// TIA Portal project "SimLogic" (V15)

(* hardware
DEVICE "S71500/ET200MP station_1"  S7-1500 station
   slot 0: "Rail_0"  Rack  6ES7 590-1***0-0AA0
   slot 1: "PLC_1"  CPU 1511-1 PN  6ES7 511-1AK00-0AB0  V1.8
      slot 3: "CPU display_1"  6ES7591-1AA00-0AA0
DEVICE "PC-System_1"  SIMATIC PC station
   slot 0: "SIMATIC PC station"  Rail  SIMATIC PC-Station  V1.0
      slot 125: "Stationmanager"  Station_Manager  V6.0.4
   slot 1: "HMI_RT_1"  WinCC RT Advanced  6AV2 104-0xxxx-xxxx  15.0.0.0
      slot 33792: "Host interface"  Host interface
   slot 2: "IE general_1"  IE General  IE_CP  V8.2.0
*)

// ===== PLC "PLC_1"  CPU 1511-1 PN =====

VAR_GLOBAL   // PLC tag table "Default tag table"
   "Brake_Out" AT %M0.0 : Bool;
   "Baffle_Out" AT %MW18 : Int;
   "RPM_In" AT %MW2 : Int;
   "OilTemp_In" AT %MW4 : Int;
   "Baffle_En" AT %M0.1 : Bool;
   "Current_In" AT %MW6 : Int;
   "OilPumpVFDsp_Out" AT %MW8 : Int;
   "OilPumpVFDen_Out" AT %M0.2 : Bool;
   "OilFlow_In" AT %MW10 : Int;
   "PB_LAD" AT %M0.3 : Bool;
   "ONS" AT %M0.4 : Bool;
   "PROGLANG" AT %MW12 : Int;
   "ONS3" AT %M0.5 : Bool;
   "ONS2" AT %M0.6 : Bool;
   "ONS1" AT %M0.7 : Bool;
   "PB_FBD" AT %M1.0 : Bool;
   "PB_SCL" AT %M1.1 : Bool;
   "PB_STL" AT %M1.2 : Bool;
   "AlarmHorn_out" AT %M1.3 : Bool;
   "stationInterlock_out" AT %M1.4 : Bool;
   "input_max" AT %MD14 : DInt;
   "OilpumpVFD_pct" AT %MW20 : Int;
   "baffle_pct" AT %MW22 : Int;
   "OiltempSV" AT %MW24 : Int;
   "OilflowSV" AT %MW26 : Int;
   "RPMout_SV" AT %MW28 : Int;
   "curentout_SV" AT %MW30 : Int;
   "oilpumpVFDoff_pb" AT %M1.5 : Bool;
   "oilpumpVFDon_pb" AT %M1.6 : Bool;
   "oilpumpVFDauto_pb" AT %M1.7 : Bool;
   "brakeoff_pb" AT %M34.0 : Bool;
   "brakeon_pb" AT %M34.1 : Bool;
   "brakeauto_pb" AT %M34.2 : Bool;
   "brakeHOA_status" AT %MW36 : Int;
   "alarmhornoff_pb" AT %M34.3 : Bool;
   "alarmhornon_pb" AT %M34.4 : Bool;
   "alarmhornauto_pb" AT %M34.5 : Bool;
   "alarmhornHOA_status" AT %MW38 : Int;
   "stationinterlockoff_pb" AT %M34.6 : Bool;
   "stationinterlockon_pb" AT %M34.7 : Bool;
   "stationinterlockauto_pb" AT %M35.0 : Bool;
   "stationinterlockHOA_status" AT %MW40 : Int;
   "oilpumpVFD_ctrl" AT %M35.1 : Bool;
   "brake_ctrl" AT %M35.2 : Bool;
   "alarmhorn_ctrl" AT %M35.3 : Bool;
   "stationinterlock_ctrl" AT %M35.4 : Bool;
   "oillowflow_SP" AT %MW44 : Int;
   "Alarm_reset" AT %M35.5 : Bool;
   "oillowflowdelay_SP" AT %MW46 : Int;
   "OI-LO-FL-AL-TRI" AT %M35.6 : Bool;
   "oillowflow_notify" AT %M48.0 : Bool;
   "alarm_rst_notify" AT %M48.1 : Bool;
   "overcurrent_SP" AT %MW50 : Int;
   "overcurrentdelya_SP" AT %MW54 : Int;
   "OV-CRNT-AL-TRI" AT %M48.2 : Bool;
   "overcurrent_notify" AT %M48.4 : Bool;
   "oilhighftempdelay_SP" AT %MW56 : Int;
   "oilhightemp_sp" AT %MW60 : Int;
   "OI-HI-TP-AL-TRI" AT %M48.5 : Bool;
   "oilhightemp_alarm" AT %M48.6 : Bool;
   "oilhightemp_notify" AT %M48.7 : Bool;
   "rotoroverspeeddelay_SP" AT %MW62 : Int;
   "RPM_SP" AT %MW66 : Int;
   "oiLtemp" AT %MW68 : Int;
   "RPM-TRI" AT %M49.0 : Bool;
   "RPM_notify" AT %M49.2 : Bool;
   "oilhighflowdelay_SP" AT %MW58 : Int;
   "oilhighflow_SP" AT %MW70 : Int;
   "OI-HI-FL-AL-TRI" AT %M49.3 : Bool;
   "oilhighflow_notify" AT %M49.5 : Bool;
   "brakefailuredelay_SP" AT %MW72 : Int;
   "brakefailure_trigger" AT %M49.7 : Bool;
   "brakefailure_notify" AT %M74.0 : Bool;
   "E-STOP" AT %M74.1 : Bool;
   "E_STOP_TRI" AT %M74.2 : Bool;
   "E-STOP_ALARM" AT %M74.3 : Bool;
   "E_STOP_NOTIFY" AT %M74.4 : Bool;
   "Tag_1" AT %T2 : Timer;
   "baffleHOA_status" AT %MW42 : Int;
   "baffle_ctrl" AT %M52.0 : Bool;
   "baffleauto_pb" AT %M52.1 : Bool;
   "baffleon_pb" AT %M52.2 : Bool;
   "warmup_mode" AT %M52.3 : Bool;
   "warmupRPM_SPIN" AT %MW64 : Int;
   "warmupVFD_SPIN" AT %MW78 : Int;
   "warmupoiltemp_SP" AT %MW82 : Int;
   "warmupoiltempdelay_sp" AT %MW84 : Int;
   "warmup_transition" AT %M52.4 : Bool;
   "current" AT %MW86 : Int;
   "bafflePIDin" AT %MW88 : Int;
   "rpm" AT %MW90 : Int;
   "stabilize_mode" AT %M52.5 : Bool;
   "stabilizekw_SPIN" AT %MW92 : Int;
   "bafflePIDsp" AT %MW94 : Int;
   "Tag_2" AT %T1 : Timer;
   "stablizemode_delay" AT %MW96 : Int;
   "stabilize_transition" AT %M52.6 : Bool;
   "generation_mode" AT %M52.7 : Bool;
   "systemstart_pb" AT %M53.0 : Bool;
   "startsequence" AT %M53.2 : Bool;
   "systemstop_pb" AT %M53.3 : Bool;
   "generation_transition" AT %M53.4 : Bool;
   "cooldown_mode" AT %M53.1 : Bool;
   "cooldownRPM_SPIN" AT %MW98 : Int;
   "cooldowndelaysp" AT %MW100 : Int;
   "cooldown_transition" AT %M53.5 : Bool;
   "cooldownoiltemp_sp" AT %MW102 : Int;
   "idlemode" AT %M53.6 : Bool;
   "faultmode" AT %M53.7 : Bool;
   "idlemode_transition" AT %M74.5 : Bool;
   "warmupVFD_SPOUT" AT %MW76 : Int;
   "Tag_3" AT %T11 : Timer;
   "sequencerunning" AT %M74.6 : Bool;
   "ons5" AT %M74.7 : Bool;
   "init_sequence" AT %M75.0 : Bool;
   "ons6" AT %M75.1 : Bool;
   "VFD_sp" AT %MW80 : Int;
   "HOAoverridevfd_sp" AT %MW104 : Int;
   "baffleoff_pb" AT %M75.2 : Bool;
   "ons7" AT %M75.3 : Bool;
   "ons8" AT %M75.4 : Bool;
   "ons9" AT %M75.5 : Bool;
   "bafflemanual" AT %M75.6 : Bool;
   "bafflemanualsp" AT %MD106 : Real;
   "ons10" AT %M75.7 : Bool;
   "ons11" AT %M110.0 : Bool;
   "vfdon_pb" AT %M110.1 : Bool;
   "ons12" AT %M110.2 : Bool;
   "ons13" AT %M110.3 : Bool;
   "ons14" AT %M110.4 : Bool;
   "ons15" AT %M110.5 : Bool;
   "ons16" AT %M110.6 : Bool;
   "vfdoff_pb" AT %M110.7 : Bool;
   "vfdauto_pb" AT %M111.0 : Bool;
   "vfdmanualsp" AT %MD114 : Real;
   "vfdmanual" AT %M111.1 : Bool;
   "bafflePID_on" AT %M111.2 : Bool;
   "oilpumpvfdpid_on" AT %M111.3 : Bool;
   "vfdHOA_status" AT %MW112 : Int;
   "fullautobit" AT %M111.4 : Bool;
   "1minutedonebit" AT %M32.0 : Bool;
   "minutesdonebit" AT %M32.1 : Bool;
   "HM_MINUTES" AT %MW118 : Int;
   "minutesreset" AT %M111.7 : Bool;
   "hoursreset" AT %M126.0 : Bool;
   "hoursdonebit" AT %M32.2 : Bool;
   "HM_HOURS" AT %MW120 : Int;
   "HM_DAYS" AT %MW122 : Int;
   "daysdonebit" AT %M32.3 : Bool;
   "daysreset" AT %M32.4 : Bool;
   "resethourmeter" AT %M32.5 : Bool;
   "resettrigger" AT %M111.6 : Bool;
   "initailminreset" AT %M32.6 : Bool;
   "SIMON" AT %M32.7 : Bool;
   "alamhorn_ctrl" AT %M33.0 : Bool;
   "oillowflow_alarm" AT %M33.1 : Bool;
   "overcurrent_alarm" AT %M33.2 : Bool;
   "RPM_ALM" AT %M33.3 : Bool;
   "oilhighflow_alarm" AT %M33.4 : Bool;
   "brakefailure_alarm" AT %M33.5 : Bool;
END_VAR

DATA_BLOCK "SimLogic_DB"   // DB1
{ S7_Optimized_Access := 'TRUE' }
VERSION : 0.1
// stored: InstanceOfName SimLogic
"SimLogic"
BEGIN
END_DATA_BLOCK

DATA_BLOCK "IO_LAD_DB"   // DB2
{ S7_Optimized_Access := 'TRUE' }
VERSION : 0.1
// stored: InstanceOfName IO_LAD
"IO_LAD"
BEGIN
END_DATA_BLOCK

DATA_BLOCK "IO_FBD_DB"   // DB4
{ S7_Optimized_Access := 'TRUE' }
VERSION : 0.1
// stored: InstanceOfName IO_FBD
"IO_FBD"
BEGIN
END_DATA_BLOCK

DATA_BLOCK "IO_SCL_DB"   // DB5
{ S7_Optimized_Access := 'TRUE' }
VERSION : 0.1
// stored: InstanceOfName IO_SCL
"IO_SCL"
BEGIN
END_DATA_BLOCK

DATA_BLOCK "IO_STL_DB"   // DB6
{ S7_Optimized_Access := 'TRUE' }
VERSION : 0.1
// stored: InstanceOfName IO_STL
"IO_STL"
BEGIN
END_DATA_BLOCK

DATA_BLOCK "HOA_LAD_DB"   // DB7
{ S7_Optimized_Access := 'TRUE' }
VERSION : 0.1
// stored: InstanceOfName HOA_LAD
"HOA_LAD"
BEGIN
END_DATA_BLOCK

DATA_BLOCK "HOA_FBD_DB"   // DB8
{ S7_Optimized_Access := 'TRUE' }
VERSION : 0.1
// stored: InstanceOfName HOA_FBD
"HOA_FBD"
BEGIN
END_DATA_BLOCK

DATA_BLOCK "HOA_SCL_DB"   // DB9
{ S7_Optimized_Access := 'TRUE' }
VERSION : 0.1
// stored: InstanceOfName HOA_SCL
"HOA_SCL"
BEGIN
END_DATA_BLOCK

DATA_BLOCK "HOA_STL_DB"   // DB10
{ S7_Optimized_Access := 'TRUE' }
VERSION : 0.1
// stored: InstanceOfName HOA_STL
"HOA_STL"
BEGIN
END_DATA_BLOCK

DATA_BLOCK "ALARM_LAD_DB"   // DB11
{ S7_Optimized_Access := 'TRUE' }
VERSION : 0.1
// stored: InstanceOfName ALARM_LAD
"ALARM_LAD"
BEGIN
END_DATA_BLOCK

DATA_BLOCK "ALARM_FBD_DB"   // DB12
{ S7_Optimized_Access := 'TRUE' }
VERSION : 0.1
// stored: InstanceOfName ALARM_FBD
"ALARM_FBD"
BEGIN
END_DATA_BLOCK

DATA_BLOCK "ALARM_SCL_DB"   // DB13
{ S7_Optimized_Access := 'TRUE' }
VERSION : 0.1
// stored: InstanceOfName ALARM_SCL
"ALARM_SCL"
BEGIN
END_DATA_BLOCK

DATA_BLOCK "ALARM_STL_DB"   // DB14
{ S7_Optimized_Access := 'TRUE' }
VERSION : 0.1
// stored: InstanceOfName ALARM_STL
"ALARM_STL"
BEGIN
END_DATA_BLOCK

DATA_BLOCK "MODES_LAD_DB"   // DB28
{ S7_Optimized_Access := 'TRUE' }
VERSION : 0.1
// stored: InstanceOfName MODES_LAD
"MODES_LAD"
BEGIN
END_DATA_BLOCK

DATA_BLOCK "MODES_FBD_DB"   // DB41
{ S7_Optimized_Access := 'TRUE' }
VERSION : 0.1
// stored: InstanceOfName MODES_FBD
"MODES_FBD"
BEGIN
END_DATA_BLOCK

DATA_BLOCK "MODES_SCL_DB"   // DB44
{ S7_Optimized_Access := 'TRUE' }
VERSION : 0.1
// stored: InstanceOfName MODES_SCL
"MODES_SCL"
BEGIN
END_DATA_BLOCK

DATA_BLOCK "MODES_STL_DB"   // DB45
{ S7_Optimized_Access := 'TRUE' }
VERSION : 0.1
// stored: InstanceOfName MODES_STL
"MODES_STL"
BEGIN
END_DATA_BLOCK

DATA_BLOCK "Sequence_DB"   // DB57
{ S7_Optimized_Access := 'TRUE' }
VERSION : 0.1
// stored: InstanceOfName Sequence
"Sequence"
BEGIN
END_DATA_BLOCK

DATA_BLOCK "Hourmeter_LAD_DB"   // DB61
{ S7_Optimized_Access := 'TRUE' }
VERSION : 0.1
// stored: InstanceOfName Hourmeter_LAD
"Hourmeter_LAD"
BEGIN
END_DATA_BLOCK

DATA_BLOCK "HOURMETER_FBD_DB"   // DB62
{ S7_Optimized_Access := 'TRUE' }
VERSION : 0.1
// stored: InstanceOfName HOURMETER_FBD
"HOURMETER_FBD"
BEGIN
END_DATA_BLOCK

DATA_BLOCK "HOURMETER_SCL_DB"   // DB63
{ S7_Optimized_Access := 'TRUE' }
VERSION : 0.1
// stored: InstanceOfName HOURMETER_SCL
"HOURMETER_SCL"
BEGIN
END_DATA_BLOCK

DATA_BLOCK "HOURMETER_STL_DB"   // DB64
{ S7_Optimized_Access := 'TRUE' }
VERSION : 0.1
// stored: InstanceOfName HOURMETER_STL
"HOURMETER_STL"
BEGIN
END_DATA_BLOCK

// folder: System blocks/Program resources

DATA_BLOCK "IEC_Timer_0_DB_25"   // DB3
{ S7_Optimized_Access := 'TRUE' }
AUTHOR : Simatic
FAMILY : IEC
NAME : IEC_TMR
VERSION : 1.0
// stored: InstanceOfName IEC_TIMER
"IEC_TIMER"
BEGIN
END_DATA_BLOCK

DATA_BLOCK "IEC_Timer_0_DB_1"   // DB15
{ S7_Optimized_Access := 'TRUE' }
AUTHOR : Simatic
FAMILY : IEC
NAME : IEC_TMR
VERSION : 1.0
// stored: InstanceOfName IEC_TIMER
"IEC_TIMER"
BEGIN
END_DATA_BLOCK

DATA_BLOCK "IEC_Timer_0_DB_2"   // DB16
{ S7_Optimized_Access := 'TRUE' }
AUTHOR : Simatic
FAMILY : IEC
NAME : IEC_TMR
VERSION : 1.0
// stored: InstanceOfName IEC_TIMER
"IEC_TIMER"
BEGIN
END_DATA_BLOCK

DATA_BLOCK "IEC_Timer_0_DB"   // DB17
{ S7_Optimized_Access := 'TRUE' }
AUTHOR : Simatic
FAMILY : IEC
NAME : IEC_TMR
VERSION : 1.0
// stored: InstanceOfName IEC_TIMER
"IEC_TIMER"
BEGIN
END_DATA_BLOCK

DATA_BLOCK "IEC_Timer_0_DB_3"   // DB18
{ S7_Optimized_Access := 'TRUE' }
AUTHOR : Simatic
FAMILY : IEC
NAME : IEC_TMR
VERSION : 1.0
// stored: InstanceOfName IEC_TIMER
"IEC_TIMER"
BEGIN
END_DATA_BLOCK

DATA_BLOCK "IEC_Timer_0_DB_4"   // DB19
{ S7_Optimized_Access := 'TRUE' }
AUTHOR : Simatic
FAMILY : IEC
NAME : IEC_TMR
VERSION : 1.0
// stored: InstanceOfName IEC_TIMER
"IEC_TIMER"
BEGIN
END_DATA_BLOCK

DATA_BLOCK "IEC_Timer_0_DB_5"   // DB20
{ S7_Optimized_Access := 'TRUE' }
AUTHOR : Simatic
FAMILY : IEC
NAME : IEC_TMR
VERSION : 1.0
// stored: InstanceOfName IEC_TIMER
"IEC_TIMER"
BEGIN
END_DATA_BLOCK

DATA_BLOCK "IEC_Timer_0_DB_6"   // DB21
{ S7_Optimized_Access := 'TRUE' }
AUTHOR : Simatic
FAMILY : IEC
NAME : IEC_TMR
VERSION : 1.0
// stored: InstanceOfName IEC_TIMER
"IEC_TIMER"
BEGIN
END_DATA_BLOCK

DATA_BLOCK "IEC_Timer_0_DB_7"   // DB22
{ S7_Optimized_Access := 'TRUE' }
AUTHOR : Simatic
FAMILY : IEC
NAME : IEC_TMR
VERSION : 1.0
// stored: InstanceOfName IEC_TIMER
"IEC_TIMER"
BEGIN
END_DATA_BLOCK

DATA_BLOCK "IEC_Timer_0_DB_8"   // DB23
{ S7_Optimized_Access := 'TRUE' }
AUTHOR : Simatic
FAMILY : IEC
NAME : IEC_TMR
VERSION : 1.0
// stored: InstanceOfName IEC_TIMER
"IEC_TIMER"
BEGIN
END_DATA_BLOCK

DATA_BLOCK "IEC_Timer_0_DB_9"   // DB24
{ S7_Optimized_Access := 'TRUE' }
AUTHOR : Simatic
FAMILY : IEC
NAME : IEC_TMR
VERSION : 1.0
// stored: InstanceOfName IEC_TIMER
"IEC_TIMER"
BEGIN
END_DATA_BLOCK

DATA_BLOCK "IEC_Timer_0_DB_10"   // DB25
{ S7_Optimized_Access := 'TRUE' }
AUTHOR : Simatic
FAMILY : IEC
NAME : IEC_TMR
VERSION : 1.0
// stored: InstanceOfName IEC_TIMER
"IEC_TIMER"
BEGIN
END_DATA_BLOCK

DATA_BLOCK "IEC_Timer_0_DB_11"   // DB26
{ S7_Optimized_Access := 'TRUE' }
AUTHOR : Simatic
FAMILY : IEC
NAME : IEC_TMR
VERSION : 1.0
// stored: InstanceOfName IEC_TIMER
"IEC_TIMER"
BEGIN
END_DATA_BLOCK

DATA_BLOCK "IEC_Timer_0_DB_12"   // DB27
{ S7_Optimized_Access := 'TRUE' }
AUTHOR : Simatic
FAMILY : IEC
NAME : IEC_TMR
VERSION : 1.0
// stored: InstanceOfName IEC_TIMER
"IEC_TIMER"
BEGIN
END_DATA_BLOCK

DATA_BLOCK "IEC_Timer_0_DB_14"   // DB29
{ S7_Optimized_Access := 'TRUE' }
AUTHOR : Simatic
FAMILY : IEC
NAME : IEC_TMR
VERSION : 1.0
// stored: InstanceOfName IEC_TIMER
"IEC_TIMER"
BEGIN
END_DATA_BLOCK

DATA_BLOCK "IEC_Timer_0_DB_15"   // DB30
{ S7_Optimized_Access := 'TRUE' }
AUTHOR : Simatic
FAMILY : IEC
NAME : IEC_TMR
VERSION : 1.0
// stored: InstanceOfName IEC_TIMER
"IEC_TIMER"
BEGIN
END_DATA_BLOCK

DATA_BLOCK "IEC_Timer_0_DB_16"   // DB31
{ S7_Optimized_Access := 'TRUE' }
AUTHOR : Simatic
FAMILY : IEC
NAME : IEC_TMR
VERSION : 1.0
// stored: InstanceOfName IEC_TIMER
"IEC_TIMER"
BEGIN
END_DATA_BLOCK

DATA_BLOCK "IEC_Timer_0_DB_17"   // DB32
{ S7_Optimized_Access := 'TRUE' }
AUTHOR : Simatic
FAMILY : IEC
NAME : IEC_TMR
VERSION : 1.0
// stored: InstanceOfName IEC_TIMER
"IEC_TIMER"
BEGIN
END_DATA_BLOCK

DATA_BLOCK "IEC_Timer_0_DB_18"   // DB33
{ S7_Optimized_Access := 'TRUE' }
AUTHOR : Simatic
FAMILY : IEC
NAME : IEC_TMR
VERSION : 1.0
// stored: InstanceOfName IEC_TIMER
"IEC_TIMER"
BEGIN
END_DATA_BLOCK

DATA_BLOCK "IEC_Timer_0_DB_19"   // DB34
{ S7_Optimized_Access := 'TRUE' }
AUTHOR : Simatic
FAMILY : IEC
NAME : IEC_TMR
VERSION : 1.0
// stored: InstanceOfName IEC_TIMER
"IEC_TIMER"
BEGIN
END_DATA_BLOCK

DATA_BLOCK "IEC_Timer_0_DB_20"   // DB35
{ S7_Optimized_Access := 'TRUE' }
AUTHOR : Simatic
FAMILY : IEC
NAME : IEC_TMR
VERSION : 1.0
// stored: InstanceOfName IEC_TIMER
"IEC_TIMER"
BEGIN
END_DATA_BLOCK

DATA_BLOCK "IEC_Timer_0_DB_21"   // DB36
{ S7_Optimized_Access := 'TRUE' }
AUTHOR : Simatic
FAMILY : IEC
NAME : IEC_TMR
VERSION : 1.0
// stored: InstanceOfName IEC_TIMER
"IEC_TIMER"
BEGIN
END_DATA_BLOCK

DATA_BLOCK "IEC_Timer_0_DB_22"   // DB37
{ S7_Optimized_Access := 'TRUE' }
AUTHOR : Simatic
FAMILY : IEC
NAME : IEC_TMR
VERSION : 1.0
// stored: InstanceOfName IEC_TIMER
"IEC_TIMER"
BEGIN
END_DATA_BLOCK

DATA_BLOCK "IEC_Timer_0_DB_23"   // DB38
{ S7_Optimized_Access := 'TRUE' }
AUTHOR : Simatic
FAMILY : IEC
NAME : IEC_TMR
VERSION : 1.0
// stored: InstanceOfName IEC_TIMER
"IEC_TIMER"
BEGIN
END_DATA_BLOCK

DATA_BLOCK "IEC_Timer_0_DB_24"   // DB39
{ S7_Optimized_Access := 'TRUE' }
AUTHOR : Simatic
FAMILY : IEC
NAME : IEC_TMR
VERSION : 1.0
// stored: InstanceOfName IEC_TIMER
"IEC_TIMER"
BEGIN
END_DATA_BLOCK

DATA_BLOCK "IEC_Timer_0_DB_26"   // DB40
{ S7_Optimized_Access := 'TRUE' }
AUTHOR : Simatic
FAMILY : IEC
NAME : IEC_TMR
VERSION : 1.0
// stored: InstanceOfName IEC_TIMER
"IEC_TIMER"
BEGIN
END_DATA_BLOCK

DATA_BLOCK "IEC_Timer_1_DB"   // DB43
{ S7_Optimized_Access := 'TRUE' }
AUTHOR : Simatic
FAMILY : IEC
NAME : IEC_TMR
VERSION : 1.0
// stored: InstanceOfName IEC_TIMER
"IEC_TIMER"
BEGIN
END_DATA_BLOCK

DATA_BLOCK "IEC_Timer_0_DB_13"   // DB46
{ S7_Optimized_Access := 'TRUE' }
AUTHOR : Simatic
FAMILY : IEC
NAME : IEC_TMR
VERSION : 1.0
// stored: InstanceOfName IEC_TIMER
"IEC_TIMER"
BEGIN
END_DATA_BLOCK

DATA_BLOCK "IEC_Timer_0_DB_27"   // DB47
{ S7_Optimized_Access := 'TRUE' }
AUTHOR : Simatic
FAMILY : IEC
NAME : IEC_TMR
VERSION : 1.0
// stored: InstanceOfName IEC_TIMER
"IEC_TIMER"
BEGIN
END_DATA_BLOCK

DATA_BLOCK "IEC_Timer_0_DB_28"   // DB48
{ S7_Optimized_Access := 'TRUE' }
AUTHOR : Simatic
FAMILY : IEC
NAME : IEC_TMR
VERSION : 1.0
// stored: InstanceOfName IEC_TIMER
"IEC_TIMER"
BEGIN
END_DATA_BLOCK

DATA_BLOCK "IEC_Timer_0_DB_29"   // DB49
{ S7_Optimized_Access := 'TRUE' }
AUTHOR : Simatic
FAMILY : IEC
NAME : IEC_TMR
VERSION : 1.0
// stored: InstanceOfName IEC_TIMER
"IEC_TIMER"
BEGIN
END_DATA_BLOCK

DATA_BLOCK "IEC_Timer_0_DB_30"   // DB50
{ S7_Optimized_Access := 'TRUE' }
AUTHOR : Simatic
FAMILY : IEC
NAME : IEC_TMR
VERSION : 1.0
// stored: InstanceOfName IEC_TIMER
"IEC_TIMER"
BEGIN
END_DATA_BLOCK

DATA_BLOCK "IEC_Timer_0_DB_31"   // DB51
{ S7_Optimized_Access := 'TRUE' }
AUTHOR : Simatic
FAMILY : IEC
NAME : IEC_TMR
VERSION : 1.0
// stored: InstanceOfName IEC_TIMER
"IEC_TIMER"
BEGIN
END_DATA_BLOCK

DATA_BLOCK "IEC_Timer_0_DB_32"   // DB52
{ S7_Optimized_Access := 'TRUE' }
AUTHOR : Simatic
FAMILY : IEC
NAME : IEC_TMR
VERSION : 1.0
// stored: InstanceOfName IEC_TIMER
"IEC_TIMER"
BEGIN
END_DATA_BLOCK

DATA_BLOCK "IEC_Timer_0_DB_33"   // DB53
{ S7_Optimized_Access := 'TRUE' }
AUTHOR : Simatic
FAMILY : IEC
NAME : IEC_TMR
VERSION : 1.0
// stored: InstanceOfName IEC_TIMER
"IEC_TIMER"
BEGIN
END_DATA_BLOCK

DATA_BLOCK "IEC_Timer_0_DB_34"   // DB54
{ S7_Optimized_Access := 'TRUE' }
AUTHOR : Simatic
FAMILY : IEC
NAME : IEC_TMR
VERSION : 1.0
// stored: InstanceOfName IEC_TIMER
"IEC_TIMER"
BEGIN
END_DATA_BLOCK

DATA_BLOCK "IEC_Timer_0_DB_35"   // DB55
{ S7_Optimized_Access := 'TRUE' }
AUTHOR : Simatic
FAMILY : IEC
NAME : IEC_TMR
VERSION : 1.0
// stored: InstanceOfName IEC_TIMER
"IEC_TIMER"
BEGIN
END_DATA_BLOCK

DATA_BLOCK "IEC_Timer_0_DB_36"   // DB56
{ S7_Optimized_Access := 'TRUE' }
AUTHOR : Simatic
FAMILY : IEC
NAME : IEC_TMR
VERSION : 1.0
// stored: InstanceOfName IEC_TIMER
"IEC_TIMER"
BEGIN
END_DATA_BLOCK

DATA_BLOCK "IEC_Timer_0_DB_37"   // DB65
{ S7_Optimized_Access := 'TRUE' }
AUTHOR : Simatic
FAMILY : IEC
NAME : IEC_TMR
VERSION : 1.0
// stored: InstanceOfName IEC_TIMER
"IEC_TIMER"
BEGIN
END_DATA_BLOCK

DATA_BLOCK "IEC_Counter_0_DB_1"   // DB67
{ S7_Optimized_Access := 'TRUE' }
AUTHOR : Simatic
FAMILY : IEC
NAME : CNTR
VERSION : 1.0
// stored: InstanceOfName IEC_COUNTER
"IEC_COUNTER"
BEGIN
END_DATA_BLOCK

DATA_BLOCK "IEC_Counter_0_DB_2"   // DB68
{ S7_Optimized_Access := 'TRUE' }
AUTHOR : Simatic
FAMILY : IEC
NAME : CNTR
VERSION : 1.0
// stored: InstanceOfName IEC_COUNTER
"IEC_COUNTER"
BEGIN
END_DATA_BLOCK

DATA_BLOCK "IEC_Timer_0_DB_38"   // DB69
{ S7_Optimized_Access := 'TRUE' }
AUTHOR : Simatic
FAMILY : IEC
NAME : IEC_TMR
VERSION : 1.0
// stored: InstanceOfName IEC_TIMER
"IEC_TIMER"
BEGIN
END_DATA_BLOCK

DATA_BLOCK "IEC_Timer_0_DB_39"   // DB71
{ S7_Optimized_Access := 'TRUE' }
AUTHOR : Simatic
FAMILY : IEC
NAME : IEC_TMR
VERSION : 1.0
// stored: InstanceOfName IEC_TIMER
"IEC_TIMER"
BEGIN
END_DATA_BLOCK

DATA_BLOCK "IEC_Counter_0_DB_4"   // DB72
{ S7_Optimized_Access := 'TRUE' }
AUTHOR : Simatic
FAMILY : IEC
NAME : CNTR
VERSION : 1.0
// stored: InstanceOfName IEC_COUNTER
"IEC_COUNTER"
BEGIN
END_DATA_BLOCK

DATA_BLOCK "IEC_Counter_0_DB_5"   // DB73
{ S7_Optimized_Access := 'TRUE' }
AUTHOR : Simatic
FAMILY : IEC
NAME : CNTR
VERSION : 1.0
// stored: InstanceOfName IEC_COUNTER
"IEC_COUNTER"
BEGIN
END_DATA_BLOCK

DATA_BLOCK "IEC_Counter_0_DB_6"   // DB74
{ S7_Optimized_Access := 'TRUE' }
AUTHOR : Simatic
FAMILY : IEC
NAME : CNTR
VERSION : 1.0
// stored: InstanceOfName IEC_COUNTER
"IEC_COUNTER"
BEGIN
END_DATA_BLOCK

DATA_BLOCK "IEC_Timer_0_DB_40"   // DB75
{ S7_Optimized_Access := 'TRUE' }
AUTHOR : Simatic
FAMILY : IEC
NAME : IEC_TMR
VERSION : 1.0
// stored: InstanceOfName IEC_TIMER
"IEC_TIMER"
BEGIN
END_DATA_BLOCK

DATA_BLOCK "IEC_Timer_0_DB_42"   // DB78
{ S7_Optimized_Access := 'TRUE' }
AUTHOR : Simatic
FAMILY : IEC
NAME : IEC_TMR
VERSION : 1.0
// stored: InstanceOfName IEC_TIMER
"IEC_TIMER"
BEGIN
END_DATA_BLOCK

DATA_BLOCK "IEC_Counter_0_DB_7"   // DB79
{ S7_Optimized_Access := 'TRUE' }
AUTHOR : Simatic
FAMILY : IEC
NAME : CNTR
VERSION : 1.0
// stored: InstanceOfName IEC_COUNTER
"IEC_COUNTER"
BEGIN
END_DATA_BLOCK

DATA_BLOCK "IEC_Counter_0_DB_8"   // DB80
{ S7_Optimized_Access := 'TRUE' }
AUTHOR : Simatic
FAMILY : IEC
NAME : CNTR
VERSION : 1.0
// stored: InstanceOfName IEC_COUNTER
"IEC_COUNTER"
BEGIN
END_DATA_BLOCK

DATA_BLOCK "IEC_Counter_0_DB_9"   // DB81
{ S7_Optimized_Access := 'TRUE' }
AUTHOR : Simatic
FAMILY : IEC
NAME : CNTR
VERSION : 1.0
// stored: InstanceOfName IEC_COUNTER
"IEC_COUNTER"
BEGIN
END_DATA_BLOCK

DATA_BLOCK "IEC_Timer_0_DB_43"   // DB82
{ S7_Optimized_Access := 'TRUE' }
AUTHOR : Simatic
FAMILY : IEC
NAME : IEC_TMR
VERSION : 1.0
// stored: InstanceOfName IEC_TIMER
"IEC_TIMER"
BEGIN
END_DATA_BLOCK

DATA_BLOCK "IEC_Timer_0_DB_44"   // DB83
{ S7_Optimized_Access := 'TRUE' }
AUTHOR : Simatic
FAMILY : IEC
NAME : IEC_TMR
VERSION : 1.0
// stored: InstanceOfName IEC_TIMER
"IEC_TIMER"
BEGIN
END_DATA_BLOCK

DATA_BLOCK "IEC_Timer_0_DB_45"   // DB84
{ S7_Optimized_Access := 'TRUE' }
AUTHOR : Simatic
FAMILY : IEC
NAME : IEC_TMR
VERSION : 1.0
// stored: InstanceOfName IEC_TIMER
"IEC_TIMER"
BEGIN
END_DATA_BLOCK

DATA_BLOCK "IEC_Counter_0_DB_10"   // DB85
{ S7_Optimized_Access := 'TRUE' }
AUTHOR : Simatic
FAMILY : IEC
NAME : CNTR
VERSION : 1.0
// stored: InstanceOfName IEC_COUNTER
"IEC_COUNTER"
BEGIN
END_DATA_BLOCK

DATA_BLOCK "IEC_Counter_0_DB_11"   // DB86
{ S7_Optimized_Access := 'TRUE' }
AUTHOR : Simatic
FAMILY : IEC
NAME : CNTR
VERSION : 1.0
// stored: InstanceOfName IEC_COUNTER
"IEC_COUNTER"
BEGIN
END_DATA_BLOCK

DATA_BLOCK "IEC_Counter_0_DB_12"   // DB87
{ S7_Optimized_Access := 'TRUE' }
AUTHOR : Simatic
FAMILY : IEC
NAME : CNTR
VERSION : 1.0
// stored: InstanceOfName IEC_COUNTER
"IEC_COUNTER"
BEGIN
END_DATA_BLOCK

// folder: (top level)

FUNCTION_BLOCK "SimLogic"   // FB1, FBD
{ S7_Optimized_Access := 'TRUE' }
VERSION : 0.1
   VAR
      "TO" : Bool;
      rpmv : Int;
      addrpmv : Bool;
      otsp : Int;
      ott : Int;
      TO1 : Bool;
      TO2 : Bool;
      be2 : Int;
      be3 : Int;
      be1 : Int;
      TO3 : Bool;
   END_VAR
   VAR_TEMP
      bf : Int;
      rpmvt : Int;
      bfr : Real;
   END_VAR
BEGIN

REGION Network 1
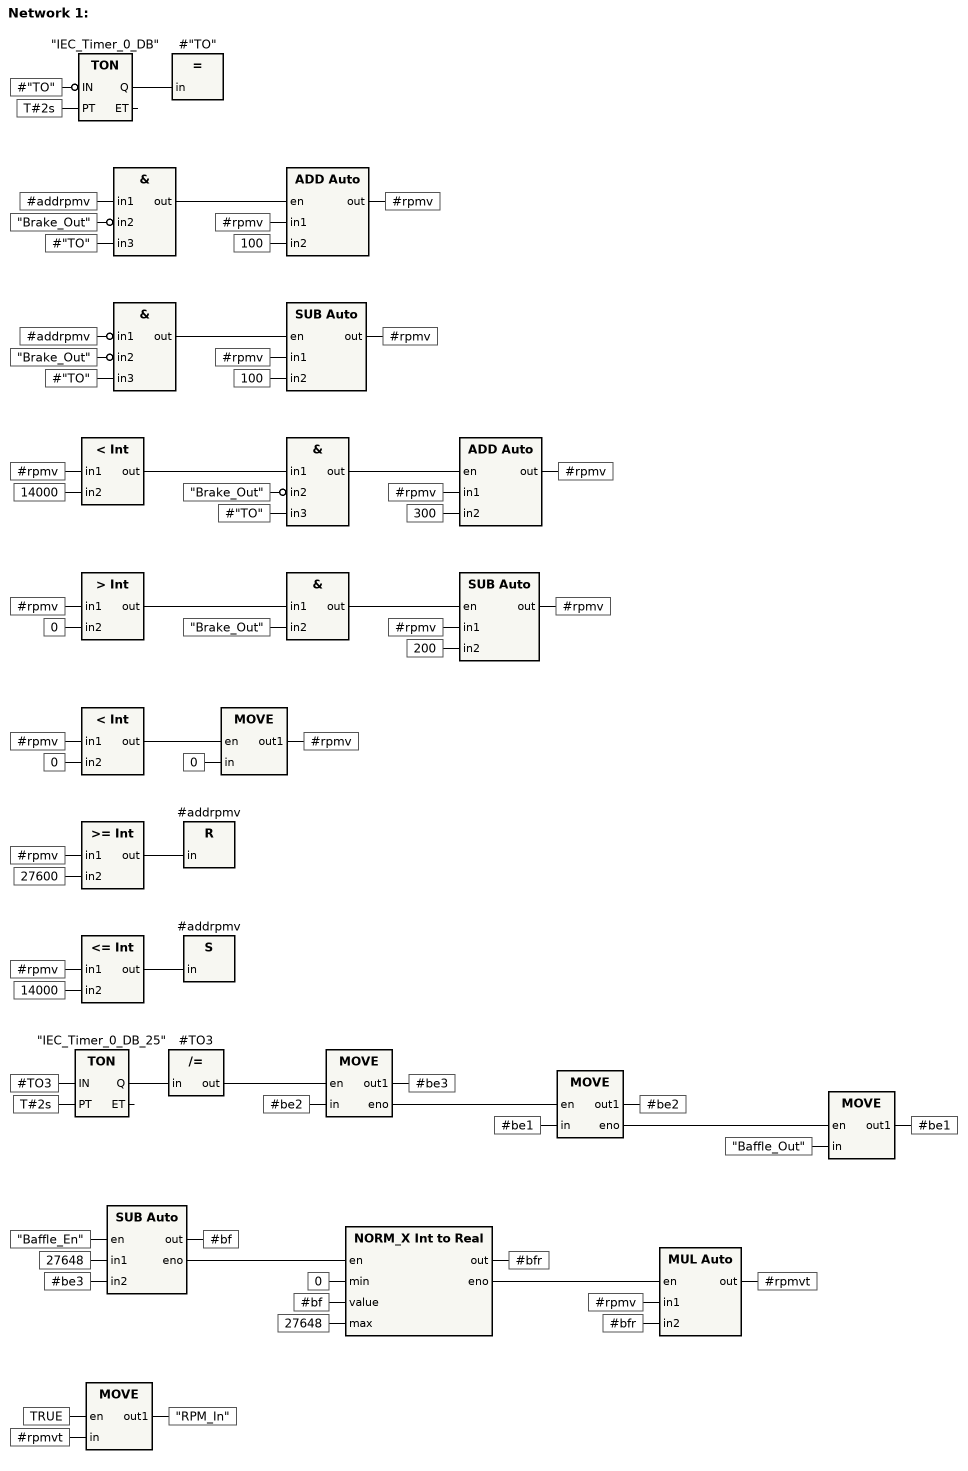
   "IEC_Timer_0_DB".TON(IN := NOT #"TO", PT := T#2s);
   #"TO" := "IEC_Timer_0_DB".Q;
   IF #addrpmv AND NOT "Brake_Out" AND #"TO" THEN #rpmv := #rpmv + 100; END_IF;
   IF NOT #addrpmv AND NOT "Brake_Out" AND #"TO" THEN #rpmv := #rpmv - 100; END_IF;
   IF (#rpmv < 14000) AND NOT "Brake_Out" AND #"TO" THEN #rpmv := #rpmv + 300; END_IF;
   IF (#rpmv > 0) AND "Brake_Out" THEN #rpmv := #rpmv - 200; END_IF;
   IF #rpmv < 0 THEN #rpmv := 0; END_IF;
   IF #rpmv >= 27600 THEN #addrpmv := FALSE; END_IF;
   IF #rpmv <= 14000 THEN #addrpmv := TRUE; END_IF;
   "IEC_Timer_0_DB_25".TON(IN := #TO3, PT := T#2s);
   #TO3 := NOT "IEC_Timer_0_DB_25".Q;
   IF "IEC_Timer_0_DB_25".Q THEN
       #be3 := #be2;
       #be2 := #be1;
       #be1 := "Baffle_Out";
   END_IF;
   IF "Baffle_En" THEN
       #bf := 27648 - #be3;
       #bfr := NORM_X(MIN := 0, VALUE := #bf, MAX := 27648);
       #rpmvt := #rpmv * #bfr;
   END_IF;
   IF TRUE THEN "RPM_In" := #rpmvt; END_IF;
END_REGION

REGION Network 2
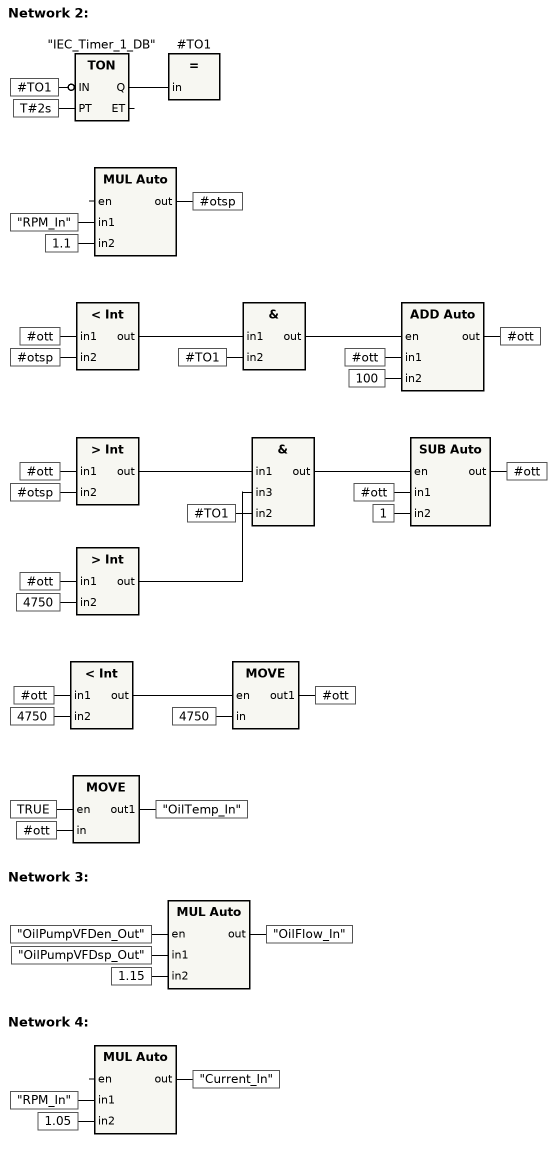
   "IEC_Timer_1_DB".TON(IN := NOT #TO1, PT := T#2s);
   #TO1 := "IEC_Timer_1_DB".Q;
   #otsp := "RPM_In" * 1.1;
   IF (#ott < #otsp) AND #TO1 THEN #ott := #ott + 100; END_IF;
   IF (#ott > #otsp) AND (#ott > 4750) AND #TO1 THEN #ott := #ott - 1; END_IF;
   IF #ott < 4750 THEN #ott := 4750; END_IF;
   IF TRUE THEN "OilTemp_In" := #ott; END_IF;
END_REGION

REGION Network 3
   IF "OilPumpVFDen_Out" THEN "OilFlow_In" := "OilPumpVFDsp_Out" * 1.15; END_IF;
END_REGION

REGION Network 4
   "Current_In" := "RPM_In" * 1.05;
END_REGION
END_FUNCTION_BLOCK

FUNCTION_BLOCK "IO_LAD"   // FB2, LAD
{ S7_Optimized_Access := 'TRUE' }
VERSION : 0.1
BEGIN

REGION Network 1
   // Digital output
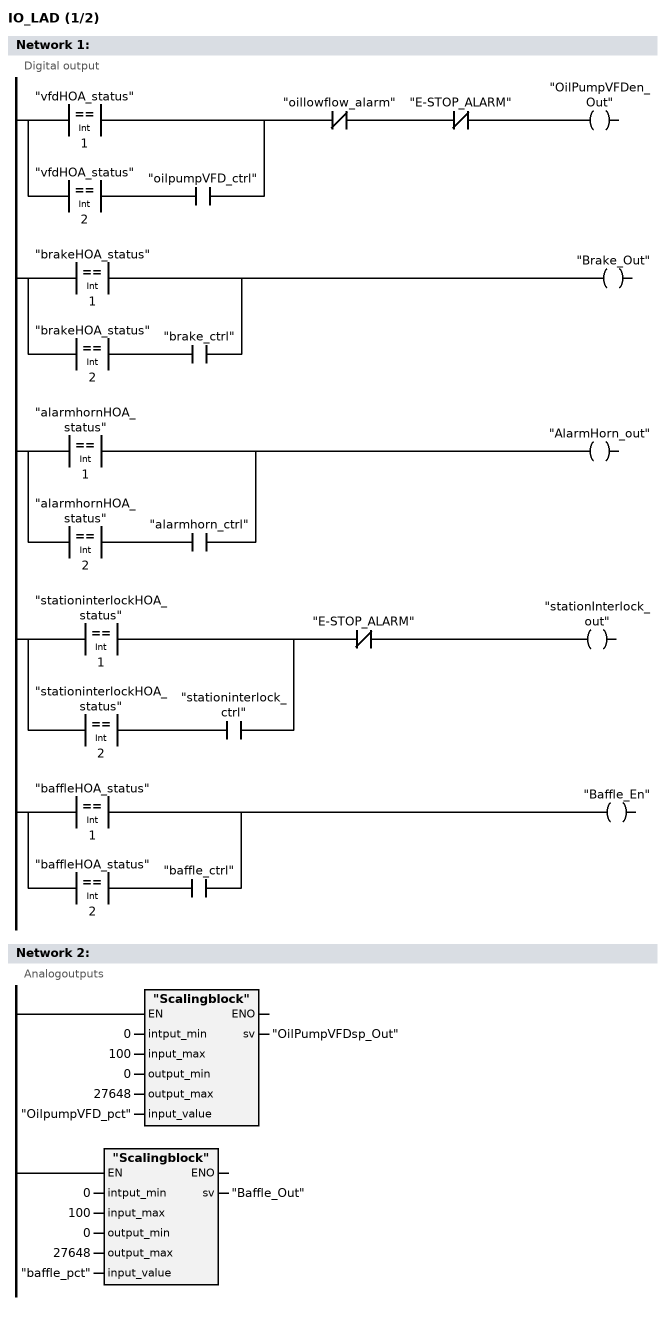
   RUNG wire#powerrail
      { S7_Templates := "SrcType := Int" } EQ_Contact(in1 := "vfdHOA_status", in2 := 1)
      wire#w1
      I_Contact( "oillowflow_alarm" )
      I_Contact( "E-STOP_ALARM" )
      Coil( "OilPumpVFDen_Out" )
   END_RUNG
   RUNG wire#powerrail
      { S7_Templates := "SrcType := Int" } EQ_Contact(in1 := "vfdHOA_status", in2 := 2)
      Contact( "oilpumpVFD_ctrl" )
   END_RUNG wire#w1
   RUNG wire#powerrail
      { S7_Templates := "SrcType := Int" } EQ_Contact(in1 := "brakeHOA_status", in2 := 1)
      wire#w2
      Coil( "Brake_Out" )
   END_RUNG
   RUNG wire#powerrail
      { S7_Templates := "SrcType := Int" } EQ_Contact(in1 := "brakeHOA_status", in2 := 2)
      Contact( "brake_ctrl" )
   END_RUNG wire#w2
   RUNG wire#powerrail
      { S7_Templates := "SrcType := Int" } EQ_Contact(in1 := "alarmhornHOA_status", in2 := 1)
      wire#w3
      Coil( "AlarmHorn_out" )
   END_RUNG
   RUNG wire#powerrail
      { S7_Templates := "SrcType := Int" } EQ_Contact(in1 := "alarmhornHOA_status", in2 := 2)
      Contact( "alarmhorn_ctrl" )
   END_RUNG wire#w3
   RUNG wire#powerrail
      { S7_Templates := "SrcType := Int" } EQ_Contact(in1 := "stationinterlockHOA_status", in2 := 1)
      wire#w4
      I_Contact( "E-STOP_ALARM" )
      Coil( "stationInterlock_out" )
   END_RUNG
   RUNG wire#powerrail
      { S7_Templates := "SrcType := Int" } EQ_Contact(in1 := "stationinterlockHOA_status", in2 := 2)
      Contact( "stationinterlock_ctrl" )
   END_RUNG wire#w4
   RUNG wire#powerrail
      { S7_Templates := "SrcType := Int" } EQ_Contact(in1 := "baffleHOA_status", in2 := 1)
      wire#w5
      Coil( "Baffle_En" )
   END_RUNG
   RUNG wire#powerrail
      { S7_Templates := "SrcType := Int" } EQ_Contact(in1 := "baffleHOA_status", in2 := 2)
      Contact( "baffle_ctrl" )
   END_RUNG wire#w5
   // the same network as SCL:
   "OilPumpVFDen_Out" := (("vfdHOA_status" = 1) OR (("vfdHOA_status" = 2) AND "oilpumpVFD_ctrl")) AND NOT "oillowflow_alarm" AND NOT "E-STOP_ALARM";
   "Brake_Out" := ("brakeHOA_status" = 1) OR (("brakeHOA_status" = 2) AND "brake_ctrl");
   "AlarmHorn_out" := ("alarmhornHOA_status" = 1) OR (("alarmhornHOA_status" = 2) AND "alarmhorn_ctrl");
   "stationInterlock_out" := (("stationinterlockHOA_status" = 1) OR (("stationinterlockHOA_status" = 2) AND "stationinterlock_ctrl")) AND NOT "E-STOP_ALARM";
   "Baffle_En" := ("baffleHOA_status" = 1) OR (("baffleHOA_status" = 2) AND "baffle_ctrl");
END_REGION

REGION Network 2
   // Analogoutputs
   RUNG wire#powerrail
      "Scalingblock"(intput_min := 0, input_max := 100, output_min := 0, output_max := 27648, input_value := "OilpumpVFD_pct", sv => "OilPumpVFDsp_Out")
   END_RUNG
   RUNG wire#powerrail
      "Scalingblock"(intput_min := 0, input_max := 100, output_min := 0, output_max := 27648, input_value := "baffle_pct", sv => "Baffle_Out")
   END_RUNG
   // the same network as SCL:
   "Scalingblock"(intput_min := 0,
                  input_max := 100,
                  output_min := 0,
                  output_max := 27648,
                  input_value := "OilpumpVFD_pct",
                  sv => "OilPumpVFDsp_Out");
   "Scalingblock"(intput_min := 0,
                  input_max := 100,
                  output_min := 0,
                  output_max := 27648,
                  input_value := "baffle_pct",
                  sv => "Baffle_Out");
END_REGION

REGION Network 3
   // Analog inputs
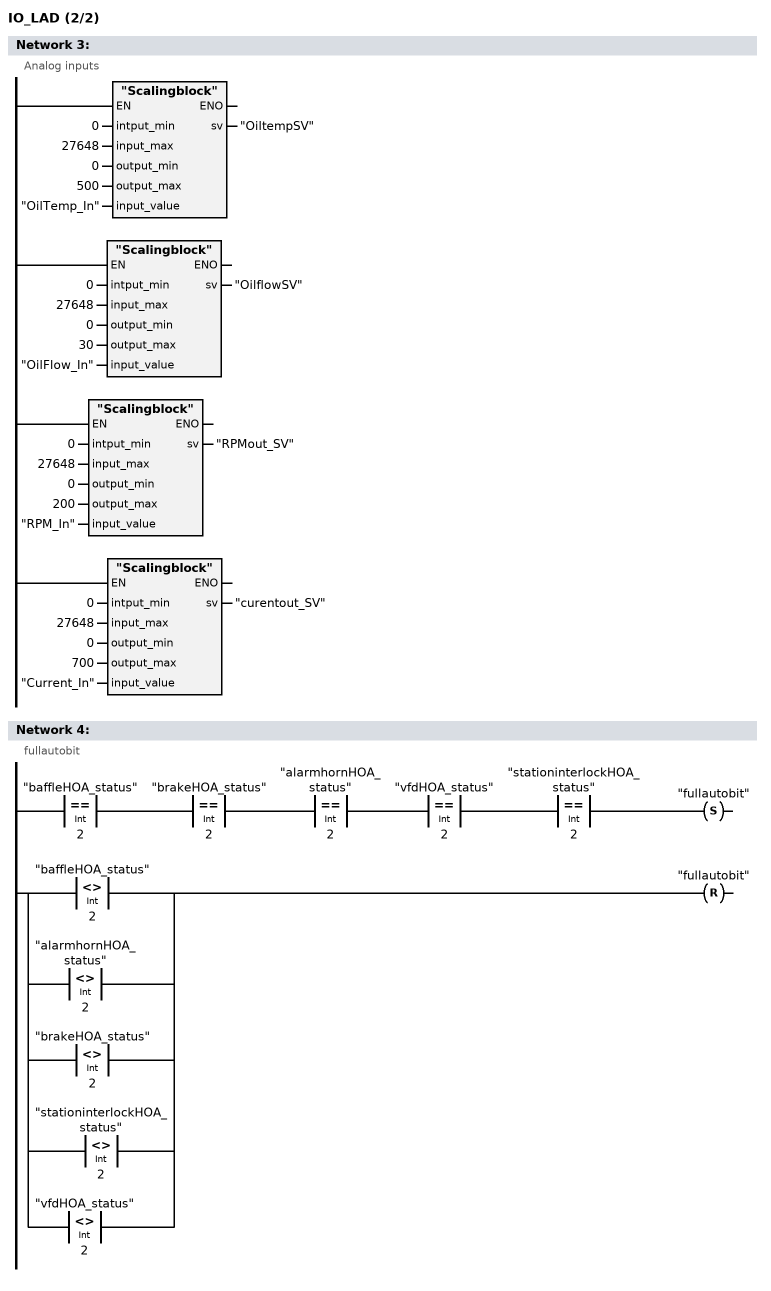
   RUNG wire#powerrail
      "Scalingblock"(intput_min := 0, input_max := 27648, output_min := 0, output_max := 500, input_value := "OilTemp_In", sv => "OiltempSV")
   END_RUNG
   RUNG wire#powerrail
      "Scalingblock"(intput_min := 0, input_max := 27648, output_min := 0, output_max := 30, input_value := "OilFlow_In", sv => "OilflowSV")
   END_RUNG
   RUNG wire#powerrail
      "Scalingblock"(intput_min := 0, input_max := 27648, output_min := 0, output_max := 200, input_value := "RPM_In", sv => "RPMout_SV")
   END_RUNG
   RUNG wire#powerrail
      "Scalingblock"(intput_min := 0, input_max := 27648, output_min := 0, output_max := 700, input_value := "Current_In", sv => "curentout_SV")
   END_RUNG
   // the same network as SCL:
   "Scalingblock"(intput_min := 0,
                  input_max := 27648,
                  output_min := 0,
                  output_max := 500,
                  input_value := "OilTemp_In",
                  sv => "OiltempSV");
   "Scalingblock"(intput_min := 0,
                  input_max := 27648,
                  output_min := 0,
                  output_max := 30,
                  input_value := "OilFlow_In",
                  sv => "OilflowSV");
   "Scalingblock"(intput_min := 0,
                  input_max := 27648,
                  output_min := 0,
                  output_max := 200,
                  input_value := "RPM_In",
                  sv => "RPMout_SV");
   "Scalingblock"(intput_min := 0,
                  input_max := 27648,
                  output_min := 0,
                  output_max := 700,
                  input_value := "Current_In",
                  sv => "curentout_SV");
END_REGION

REGION Network 4
   // fullautobit
   RUNG wire#powerrail
      { S7_Templates := "SrcType := Int" } EQ_Contact(in1 := "baffleHOA_status", in2 := 2)
      { S7_Templates := "SrcType := Int" } EQ_Contact(in1 := "brakeHOA_status", in2 := 2)
      { S7_Templates := "SrcType := Int" } EQ_Contact(in1 := "alarmhornHOA_status", in2 := 2)
      { S7_Templates := "SrcType := Int" } EQ_Contact(in1 := "vfdHOA_status", in2 := 2)
      { S7_Templates := "SrcType := Int" } EQ_Contact(in1 := "stationinterlockHOA_status", in2 := 2)
      S_Coil( "fullautobit" )
   END_RUNG
   RUNG wire#powerrail
      { S7_Templates := "SrcType := Int" } NE_Contact(in1 := "baffleHOA_status", in2 := 2)
      wire#w1
      R_Coil( "fullautobit" )
   END_RUNG
   RUNG wire#powerrail
      { S7_Templates := "SrcType := Int" } NE_Contact(in1 := "alarmhornHOA_status", in2 := 2)
   END_RUNG wire#w1
   RUNG wire#powerrail
      { S7_Templates := "SrcType := Int" } NE_Contact(in1 := "brakeHOA_status", in2 := 2)
   END_RUNG wire#w1
   RUNG wire#powerrail
      { S7_Templates := "SrcType := Int" } NE_Contact(in1 := "stationinterlockHOA_status", in2 := 2)
   END_RUNG wire#w1
   RUNG wire#powerrail
      { S7_Templates := "SrcType := Int" } NE_Contact(in1 := "vfdHOA_status", in2 := 2)
   END_RUNG wire#w1
   // the same network as SCL:
   IF ("baffleHOA_status" = 2) AND ("brakeHOA_status" = 2) AND ("alarmhornHOA_status" = 2) AND ("vfdHOA_status" = 2) AND ("stationinterlockHOA_status" = 2) THEN
       "fullautobit" := TRUE;
   END_IF;
   IF ("baffleHOA_status" <> 2) OR ("alarmhornHOA_status" <> 2) OR ("brakeHOA_status" <> 2) OR ("stationinterlockHOA_status" <> 2) OR ("vfdHOA_status" <> 2) THEN
       "fullautobit" := FALSE;
   END_IF;
END_REGION
END_FUNCTION_BLOCK

FUNCTION_BLOCK "IO_FBD"   // FB3, FBD
{ S7_Optimized_Access := 'TRUE' }
VERSION : 0.1
BEGIN

REGION Network 1
   // Digital outputs
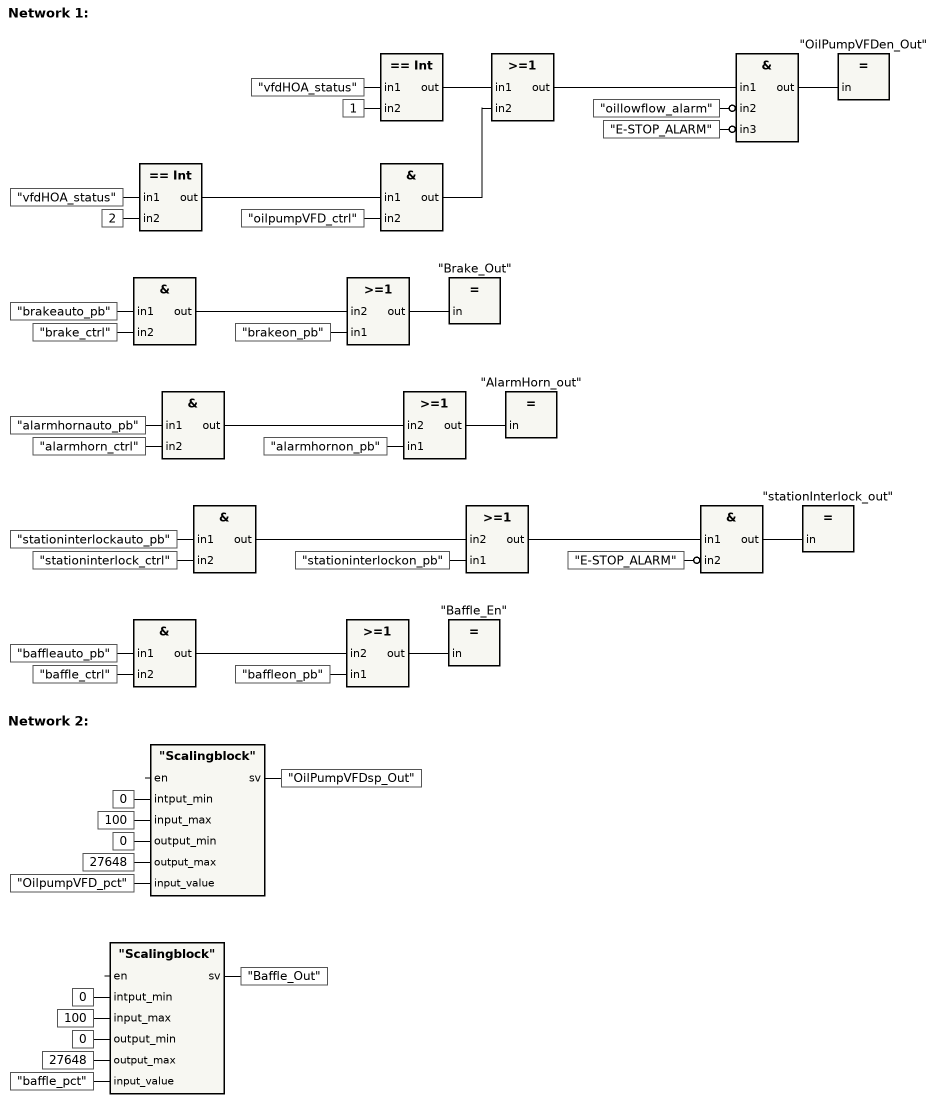
   "OilPumpVFDen_Out" := (("vfdHOA_status" = 1) OR (("vfdHOA_status" = 2) AND "oilpumpVFD_ctrl")) AND NOT "oillowflow_alarm" AND NOT "E-STOP_ALARM";
   "Brake_Out" := ("brakeauto_pb" AND "brake_ctrl") OR "brakeon_pb";
   "AlarmHorn_out" := ("alarmhornauto_pb" AND "alarmhorn_ctrl") OR "alarmhornon_pb";
   "stationInterlock_out" := (("stationinterlockauto_pb" AND "stationinterlock_ctrl") OR "stationinterlockon_pb") AND NOT "E-STOP_ALARM";
   "Baffle_En" := ("baffleauto_pb" AND "baffle_ctrl") OR "baffleon_pb";
END_REGION

REGION Network 2
   // Analogoutput
   "Scalingblock"(intput_min := 0,
                  input_max := 100,
                  output_min := 0,
                  output_max := 27648,
                  input_value := "OilpumpVFD_pct",
                  sv => "OilPumpVFDsp_Out");
   "Scalingblock"(intput_min := 0,
                  input_max := 100,
                  output_min := 0,
                  output_max := 27648,
                  input_value := "baffle_pct",
                  sv => "Baffle_Out");
END_REGION

REGION Network 3
   // analog input
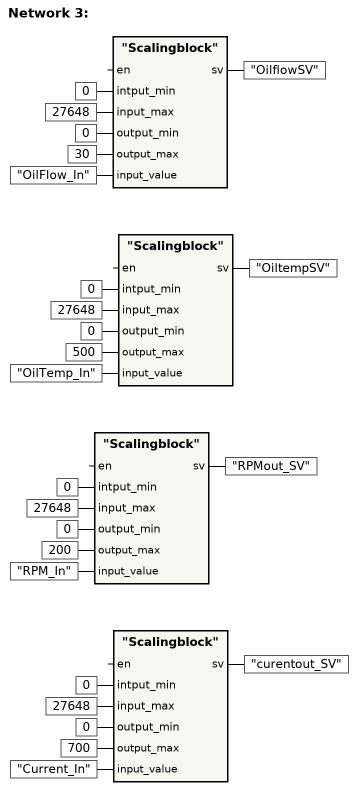
   "Scalingblock"(intput_min := 0,
                  input_max := 27648,
                  output_min := 0,
                  output_max := 30,
                  input_value := "OilFlow_In",
                  sv => "OilflowSV");
   "Scalingblock"(intput_min := 0,
                  input_max := 27648,
                  output_min := 0,
                  output_max := 500,
                  input_value := "OilTemp_In",
                  sv => "OiltempSV");
   "Scalingblock"(intput_min := 0,
                  input_max := 27648,
                  output_min := 0,
                  output_max := 200,
                  input_value := "RPM_In",
                  sv => "RPMout_SV");
   "Scalingblock"(intput_min := 0,
                  input_max := 27648,
                  output_min := 0,
                  output_max := 700,
                  input_value := "Current_In",
                  sv => "curentout_SV");
END_REGION

REGION Network 4
   // full auto bit
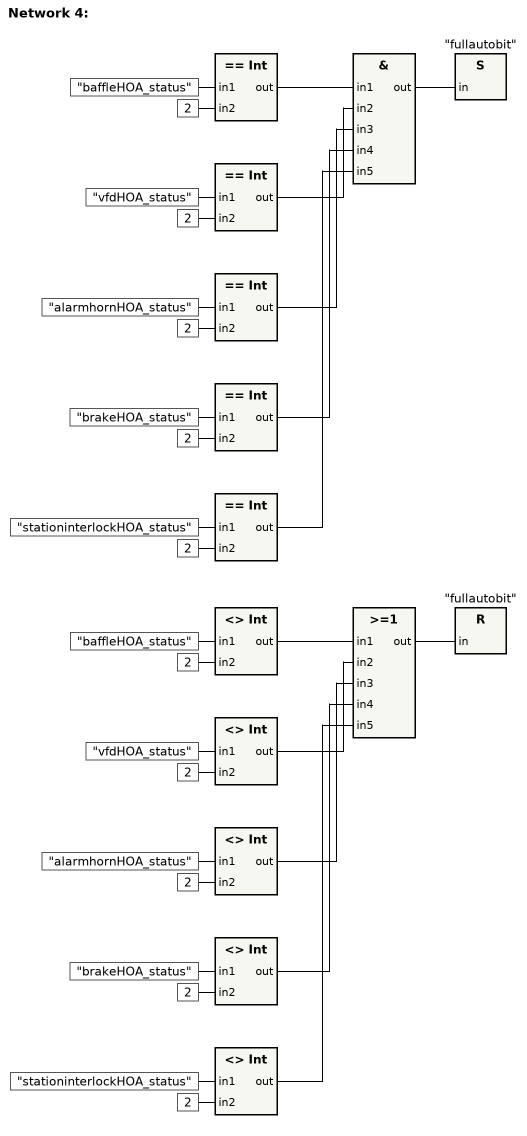
   IF ("baffleHOA_status" = 2) AND ("vfdHOA_status" = 2) AND ("alarmhornHOA_status" = 2) AND ("brakeHOA_status" = 2) AND ("stationinterlockHOA_status" = 2) THEN
       "fullautobit" := TRUE;
   END_IF;
   IF ("baffleHOA_status" <> 2) OR ("vfdHOA_status" <> 2) OR ("alarmhornHOA_status" <> 2) OR ("brakeHOA_status" <> 2) OR ("stationinterlockHOA_status" <> 2) THEN
       "fullautobit" := FALSE;
   END_IF;
END_REGION
END_FUNCTION_BLOCK

FUNCTION_BLOCK "IO_SCL"   // FB4, SCL
{ S7_Optimized_Access := 'TRUE' }
VERSION : 0.1
BEGIN
   //Digital outputs
   IF "oillowflow_alarm" OR "E-STOP_ALARM" OR "vfdHOA_status" = 0 OR ("vfdHOA_status" = 2 AND NOT "oilpumpVFD_ctrl") THEN
       "OilPumpVFDen_Out" := 0;
   END_IF;

   IF ("vfdHOA_status" = 1 OR ("vfdHOA_status" = 2 AND  "oilpumpVFD_ctrl")) AND NOT "oillowflow_alarm" AND NOT "E-STOP_ALARM" THEN
       "OilPumpVFDen_Out" := 1;
   END_IF;



   IF "brakeHOA_status" = 0 OR ( "brakeHOA_status" = 2 AND NOT "brake_ctrl") THEN
       "Brake_Out" := 0;
   END_IF;

   IF "brakeHOA_status" = 1 OR (  "brakeHOA_status" = 2 AND "brake_ctrl") THEN
        "Brake_Out" := 1;
   END_IF;


   IF "alarmhornHOA_status" = 0 OR ("alarmhornHOA_status"  = 2 AND NOT "alarmhorn_ctrl") THEN
       "AlarmHorn_out" := 0;
       END_IF;

       IF "alarmhornHOA_status"  = 1 OR ("alarmhornHOA_status"  = 2 AND "alarmhorn_ctrl") THEN
           "AlarmHorn_out" := 1;
       END_IF;

       IF "E-STOP_ALARM" OR  "stationinterlockHOA_status" = 0 OR ("stationinterlockHOA_status"  = 2 AND NOT "stationinterlock_ctrl") THEN
           "stationInterlock_out" := 0;
       END_IF;

       IF "stationinterlockHOA_status" = 1 OR ("stationinterlockHOA_status" = 2 AND "stationinterlock_ctrl") OR NOT "E-STOP_ALARM" THEN
           "stationInterlock_out" := 1;
       END_IF;

       IF "baffleHOA_status" = 0 OR ("baffleHOA_status" = 2 AND NOT "baffle_ctrl") THEN
           "Baffle_En" := 0;
       END_IF;

       IF "baffleHOA_status" = 1 OR ("baffleHOA_status" = 2 AND "baffle_ctrl") THEN
           "Baffle_En" := 1;
       END_IF;


   // Analog outputs
   "Scalingblock"(intput_min:=0,
                  input_max:=100,
                  output_min:=0,
                  output_max:=27648,
                  input_value:= "OilpumpVFD_pct",
                  sv=>"OilPumpVFDsp_Out");

   "Scalingblock"(intput_min := 0,
                  input_max := 100,
                  output_min := 0,
                  output_max := 27648,
                  input_value := "baffle_pct",
                  sv => "Baffle_Out");

   //analog inputs
   "Scalingblock"(intput_min := 0,
                  input_max := 27648,
                  output_min := 0,
                  output_max := 500,
                  input_value := "OilTemp_In",
                  sv => "OiltempSV");

   "Scalingblock"(intput_min := 0,
                  input_max := 27648,
                  output_min := 0,
                  output_max := 30,
                  input_value := "OilFlow_In",
                  sv => "OilflowSV");

   "Scalingblock"(intput_min := 0,
                  input_max := 27648,
                  output_min := 0,
                  output_max := 200,
                  input_value := "RPM_In",
                  sv => "RPMout_SV");

   "Scalingblock"(intput_min := 0,
                  input_max := 27648,
                  output_min := 0,
                  output_max := 700,
                  input_value := "Current_In",
                  sv => "curentout_SV");


   //full auto bit
   IF "baffleHOA_status" = 2 AND "alarmhornHOA_status" = 2 AND "vfdHOA_status" = 2 AND "stationinterlockHOA_status" = 2 AND "brakeHOA_status" = 2 THEN
       "fullautobit" := 1;
   ELSE
       "fullautobit" := 0;
   END_IF;
END_FUNCTION_BLOCK

FUNCTION_BLOCK "IO_STL"   // FB5, STL
{ S7_Optimized_Access := 'TRUE' }
VERSION : 0.1
BEGIN

REGION Network 1
   // digital outputs
         A     "oillowflow_alarm";
         O     "E-STOP_ALARM";
         JC    resetoilpumpvfd;
         CLR;

         L     "vfdHOA_status";
         L     0;
         ==I;
         JC    resetoilpumpvfd;
         CLR;
         L     "vfdHOA_status";
         L     1;
         ==I;
         JC    setoilpumpvfd;
         CLR;
         L     "vfdHOA_status";
         L     2;
         ==I;
         JC    autosetoilpumpvfd;



   autosetoilpumpvfd:A     "oilpumpVFD_ctrl";
         JC    setoilpumpvfd;
         JU    resetoilpumpvfd;

   setoilpumpvfd:AN    "oillowflow_alarm";
         AN    "E-STOP_ALARM";
         S     "OilPumpVFDen_Out";
         JU    Brake;

   resetoilpumpvfd:R     "OilPumpVFDen_Out";
         JU    Brake;
   //brake
   Brake:L     "brakeHOA_status";
         L     0;
         ==I;
         JC    resetbrake;
         CLR;
         L     "brakeHOA_status";
         L     1;
         ==I;
         JC    setbrake;
         CLR;
         L     "brakeHOA_status";
         L     2;
         ==I;
         JC    autosetbrake;



   autosetbrake:A     "brake_ctrl";
         JC    setbrake;
         JU    resetbrake;

   setbrake:S     "Brake_Out";
         JU    alarmhorn;

   resetbrake:R     "Brake_Out";
         JU    alarmhorn;


   //alarmhorn
   alarmhorn:L     "alarmhornHOA_status";
         L     0;
         ==I;
         JC    resetalarmhorn;
         CLR;
         L     "alarmhornHOA_status";
         L     1;
         ==I;
         JC    setalarmhorn;
         CLR;
         L     "alarmhornHOA_status";
         L     2;
         ==I;
         JC    autosetalarmhorn;



   autosetalarmhorn:A     "alarmhorn_ctrl";
         JC    setalarmhorn;
         JU    resetalarmhorn;

   setalarmhorn:S     "AlarmHorn_out";
         JU    stationinterlock;

   resetalarmhorn:R     "AlarmHorn_out";
         JU    stationinterlock;

   //stationinterlock
   stationinterlock:A     "E-STOP_ALARM";
         JC    resetstationinterlock;
         L     "stationinterlockHOA_status";
         L     0;
         ==I;
         JC    resetstationinterlock;
         CLR;
         L     "stationinterlockHOA_status";
         L     1;
         ==I;
         JC    setstationinterlock;
         CLR;
         L     "stationinterlockHOA_status";
         L     2;
         ==I;
         JC    autosetstationinterlock;



   autosetstationinterlock:A     "stationinterlock_ctrl";
         JC    setstationinterlock;
         JU    resetstationinterlock;

   setstationinterlock:AN    "E-STOP_ALARM";
         S     "stationInterlock_out";
         JU    baffle;

   resetstationinterlock:R     "stationInterlock_out";
         JU    baffle;

   // baffle

   baffle:L     "baffleHOA_status";
         L     0;
         ==I;
         JC    resetbaffle;
         CLR;
         L     "baffleHOA_status";
         L     1;
         ==I;
         JC    setbaffle;
         CLR;
         L     "baffleHOA_status";
         L     2;
         ==I;
         JC    autosetbaffle;



   autosetbaffle:A     "baffle_ctrl";
         JC    setbaffle;
         JU    resetbaffle;

   setbaffle:S     "Baffle_En";
         JU    analogoutputs;

   resetbaffle:R     "Baffle_En";
         JU    analogoutputs;

   // Analog outputs

   analogoutputs:CALL  "Scalingblock"
         ( intput_min  := 0,
           input_max   := 100,
           output_min  := 0,
           output_max  := 27648,
           input_value := "OilpumpVFD_pct",
           sv          := "OilPumpVFDsp_Out"
         );

         CALL  "Scalingblock"
         ( intput_min  := 0,
           input_max   := 100,
           output_min  := 0,
           output_max  := 27648,
           input_value := "baffle_pct",
           sv          := "Baffle_Out"
         );

   // analog inputs
   analoginputs:CALL  "Scalingblock"
         ( intput_min  := 0,
           input_max   := 27648,
           output_min  := 0,
           output_max  := 500,
           input_value := "OiltempSV",
           sv          := "OilTemp_In"
         );

         CALL  "Scalingblock"
         ( intput_min  := 0,
           input_max   := 27648,
           output_min  := 0,
           output_max  := 30,
           input_value := "OilFlow_In",
           sv          := "OilflowSV"
         );

         CALL  "Scalingblock"
         ( intput_min  := 0,
           input_max   := 27648,
           output_min  := 0,
           output_max  := 200,
           input_value := "RPM_In",
           sv          := "RPMout_SV"
         );

         CALL  "Scalingblock"
         ( intput_min  := 0,
           input_max   := 27648,
           output_min  := 0,
           output_max  := 700,
           input_value := "Current_In",
           sv          := "curentout_SV"
         );


   //fullautobit
         CLR;
         L     "baffleHOA_status";
         L     2;
         ==I;
         NOT;
         JC    resetfullauto;
         CLR;
         L     "vfdHOA_status";
         L     2;
         ==I;
         NOT;
         JC    resetfullauto;
         CLR;
         L     "alarmhornHOA_status";
         L     2;
         ==I;
         NOT;
         JC    resetfullauto;
         CLR;
         L     "brakeHOA_status";
         L     2;
         ==I;
         NOT;
         JC    resetfullauto;
         CLR;
         L     "stationinterlockHOA_status";
         L     2;
         ==I;
         NOT;
         JC    resetfullauto;
         SET;
         S     "fullautobit";
         JU    ENDOFLINE;

   resetfullauto:SET;
         NOT;
         R     "fullautobit";
         JU    ENDOFLINE;

   ENDOFLINE:BE;
END_REGION
END_FUNCTION_BLOCK

FUNCTION_BLOCK "HOA_LAD"   // FB6, LAD
{ S7_Optimized_Access := 'TRUE' }
VERSION : 0.1
   VAR
      ONSH1 : Bool;
      ONSH2 : Bool;
      ONSH3 : Bool;
      ONSH4 : Bool;
      ONSH5 : Bool;
      ONSH6 : Bool;
      ONSH9 : Bool;
      ONSH8 : Bool;
      ONSH7 : Bool;
      ONSH12 : Bool;
      ONSH11 : Bool;
      ONSH10 : Bool;
   END_VAR
   VAR_TEMP   // added for the SCL form of the ladder/FBD networks
      _w1 : Bool;
      _w2 : Bool;
      _w3 : Bool;
   END_VAR
BEGIN

REGION Network 1
   // brakeHOA
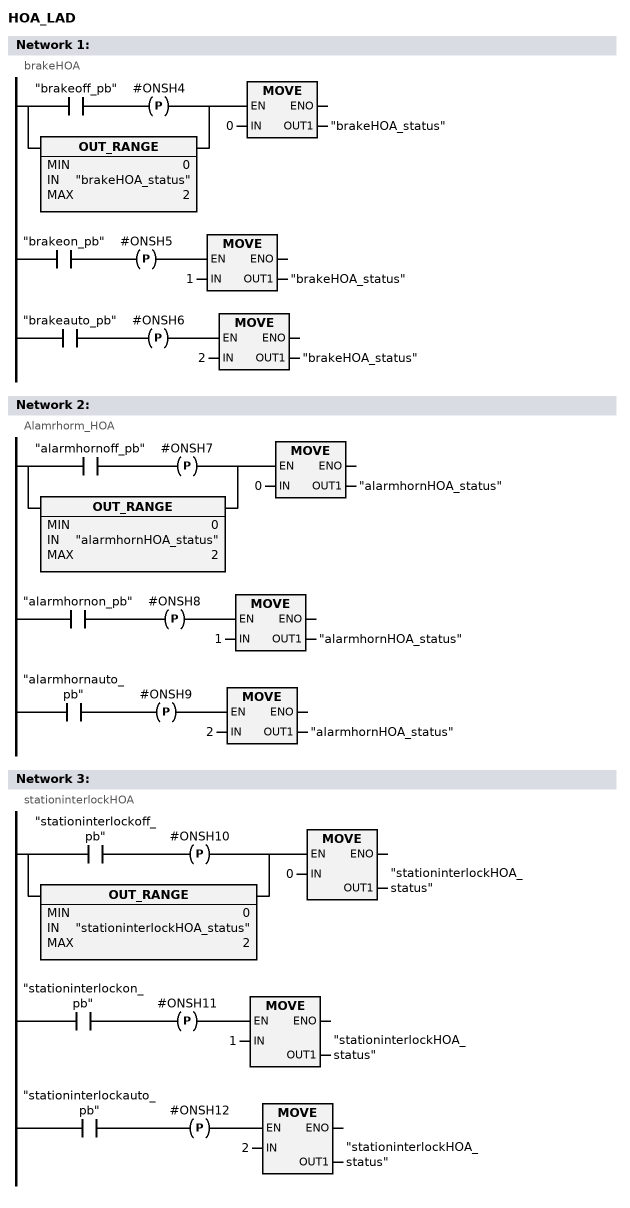
   #_w1 := "brakeoff_pb" AND NOT #ONSH4;   // rising edge
   #ONSH4 := "brakeoff_pb";
   IF #_w1 OR ("brakeHOA_status" < 0) OR ("brakeHOA_status" > 2) THEN "brakeHOA_status" := 0; END_IF;
   #_w2 := "brakeon_pb" AND NOT #ONSH5;   // rising edge
   #ONSH5 := "brakeon_pb";
   IF #_w2 THEN "brakeHOA_status" := 1; END_IF;
   #_w3 := "brakeauto_pb" AND NOT #ONSH6;   // rising edge
   #ONSH6 := "brakeauto_pb";
   IF #_w3 THEN "brakeHOA_status" := 2; END_IF;
END_REGION

REGION Network 2
   // Alamrhorm_HOA
   #_w1 := "alarmhornoff_pb" AND NOT #ONSH7;   // rising edge
   #ONSH7 := "alarmhornoff_pb";
   IF #_w1 OR ("alarmhornHOA_status" < 0) OR ("alarmhornHOA_status" > 2) THEN
       "alarmhornHOA_status" := 0;
   END_IF;
   #_w2 := "alarmhornon_pb" AND NOT #ONSH8;   // rising edge
   #ONSH8 := "alarmhornon_pb";
   IF #_w2 THEN "alarmhornHOA_status" := 1; END_IF;
   #_w3 := "alarmhornauto_pb" AND NOT #ONSH9;   // rising edge
   #ONSH9 := "alarmhornauto_pb";
   IF #_w3 THEN "alarmhornHOA_status" := 2; END_IF;
END_REGION

REGION Network 3
   // stationinterlockHOA
   #_w1 := "stationinterlockoff_pb" AND NOT #ONSH10;   // rising edge
   #ONSH10 := "stationinterlockoff_pb";
   IF #_w1 OR ("stationinterlockHOA_status" < 0) OR ("stationinterlockHOA_status" > 2) THEN
       "stationinterlockHOA_status" := 0;
   END_IF;
   #_w2 := "stationinterlockon_pb" AND NOT #ONSH11;   // rising edge
   #ONSH11 := "stationinterlockon_pb";
   IF #_w2 THEN "stationinterlockHOA_status" := 1; END_IF;
   #_w3 := "stationinterlockauto_pb" AND NOT #ONSH12;   // rising edge
   #ONSH12 := "stationinterlockauto_pb";
   IF #_w3 THEN "stationinterlockHOA_status" := 2; END_IF;
END_REGION
END_FUNCTION_BLOCK

FUNCTION_BLOCK "HOA_FBD"   // FB7, FBD
{ S7_Optimized_Access := 'TRUE' }
VERSION : 0.1
   VAR
      ONSH2 : Bool;
      ONSH3 : Bool;
      ONSH1 : Bool;
      ONSH4 : Bool;
      ONSH5 : Bool;
      ONSH6 : Bool;
      ONSH9 : Bool;
      ONSH8 : Bool;
      ONSH7 : Bool;
      ONSH12 : Bool;
      ONSH11 : Bool;
      ONSH10 : Bool;
   END_VAR
   VAR_TEMP   // added for the SCL form of the ladder/FBD networks
      _w1 : Bool;
      _w2 : Bool;
      _w3 : Bool;
   END_VAR
BEGIN

REGION Network 1
   // brake HOA
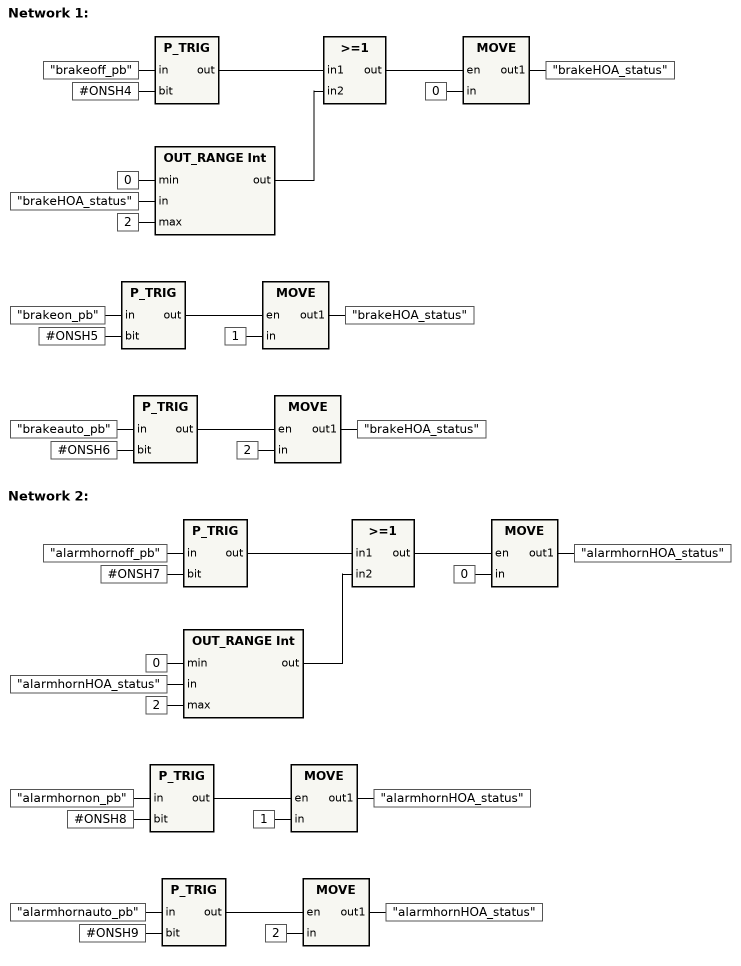
   #_w1 := "brakeoff_pb" AND NOT #ONSH4;   // rising edge
   #ONSH4 := "brakeoff_pb";
   IF #_w1 OR ("brakeHOA_status" < 0) OR ("brakeHOA_status" > 2) THEN "brakeHOA_status" := 0; END_IF;
   #_w2 := "brakeon_pb" AND NOT #ONSH5;   // rising edge
   #ONSH5 := "brakeon_pb";
   IF #_w2 THEN "brakeHOA_status" := 1; END_IF;
   #_w3 := "brakeauto_pb" AND NOT #ONSH6;   // rising edge
   #ONSH6 := "brakeauto_pb";
   IF #_w3 THEN "brakeHOA_status" := 2; END_IF;
END_REGION

REGION Network 2
   // alarmhorn HOA
   #_w1 := "alarmhornoff_pb" AND NOT #ONSH7;   // rising edge
   #ONSH7 := "alarmhornoff_pb";
   IF #_w1 OR ("alarmhornHOA_status" < 0) OR ("alarmhornHOA_status" > 2) THEN
       "alarmhornHOA_status" := 0;
   END_IF;
   #_w2 := "alarmhornon_pb" AND NOT #ONSH8;   // rising edge
   #ONSH8 := "alarmhornon_pb";
   IF #_w2 THEN "alarmhornHOA_status" := 1; END_IF;
   #_w3 := "alarmhornauto_pb" AND NOT #ONSH9;   // rising edge
   #ONSH9 := "alarmhornauto_pb";
   IF #_w3 THEN "alarmhornHOA_status" := 2; END_IF;
END_REGION

REGION Network 3
   // stationinterlock HOA
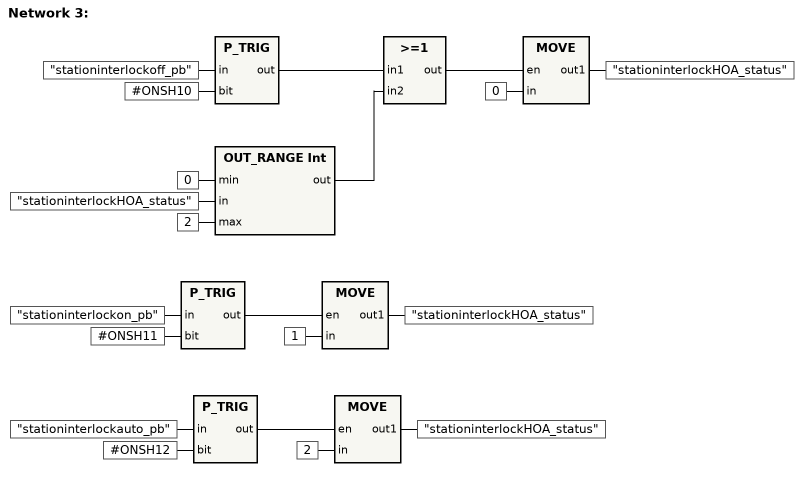
   #_w1 := "stationinterlockoff_pb" AND NOT #ONSH10;   // rising edge
   #ONSH10 := "stationinterlockoff_pb";
   IF #_w1 OR ("stationinterlockHOA_status" < 0) OR ("stationinterlockHOA_status" > 2) THEN
       "stationinterlockHOA_status" := 0;
   END_IF;
   #_w2 := "stationinterlockon_pb" AND NOT #ONSH11;   // rising edge
   #ONSH11 := "stationinterlockon_pb";
   IF #_w2 THEN "stationinterlockHOA_status" := 1; END_IF;
   #_w3 := "stationinterlockauto_pb" AND NOT #ONSH12;   // rising edge
   #ONSH12 := "stationinterlockauto_pb";
   IF #_w3 THEN "stationinterlockHOA_status" := 2; END_IF;
END_REGION
END_FUNCTION_BLOCK

FUNCTION_BLOCK "HOA_SCL"   // FB8, SCL
{ S7_Optimized_Access := 'TRUE' }
VERSION : 0.1
BEGIN


   //brake HOA 
   IF "brakeHOA_status" < 0 OR "brakeHOA_status" > 2 THEN
       "brakeHOA_status" := 0;
   END_IF;

   IF "brakeoff_pb" AND "brakeHOA_status" <> 0 THEN
       "brakeHOA_status" := 0;
   END_IF;

   IF "brakeon_pb" AND "brakeHOA_status" <> 1 THEN
       "brakeHOA_status" := 1;
   END_IF;

   IF "brakeauto_pb" AND "brakeHOA_status" <> 2 THEN
       "brakeHOA_status" := 2;
   END_IF;



   //alarmhorn HOA 
   IF "alarmhornHOA_status" < 0 OR "alarmhornHOA_status" > 2 THEN
       "alarmhornHOA_status" := 0;
   END_IF;

   IF "alarmhornoff_pb" AND "alarmhornHOA_status" <> 0 THEN
       "alarmhornHOA_status" := 0;
   END_IF;

   IF "alarmhornon_pb" AND "alarmhornHOA_status" <> 1 THEN
       "alarmhornHOA_status" := 1;
   END_IF;

   IF "alarmhornauto_pb" AND "alarmhornHOA_status" <> 2 THEN
       "alarmhornHOA_status" := 2;
   END_IF;


   //stationinterlock HOA 
   IF "stationinterlockHOA_status" < 0 OR "stationinterlockHOA_status" > 2 THEN
       "stationinterlockHOA_status" := 0;
   END_IF;

   IF "stationinterlockoff_pb" AND "stationinterlockHOA_status" <> 0 THEN
       "stationinterlockHOA_status" := 0;
   END_IF;

   IF "stationinterlockon_pb" AND "stationinterlockHOA_status" <> 1 THEN
       "stationinterlockHOA_status" := 1;
   END_IF;

   IF "stationinterlockauto_pb" AND "stationinterlockHOA_status" <> 2 THEN
       "stationinterlockHOA_status" := 2;
   END_IF;
END_FUNCTION_BLOCK

FUNCTION_BLOCK "HOA_STL"   // FB9, STL
{ S7_Optimized_Access := 'TRUE' }
VERSION : 0.1
   VAR
      ONSH1 : Bool;
      ONSH2 : Bool;
      ONSH3 : Bool;
      ONSH4 : Bool;
      ONSH5 : Bool;
      ONSH12 : Bool;
      ONSH11 : Bool;
      ONSH10 : Bool;
      ONSH9 : Bool;
      ONSH8 : Bool;
      ONSH7 : Bool;
   END_VAR
   VAR_TEMP
      ONSH6 : Bool;
   END_VAR
BEGIN

REGION Network 1



   brake:L     "brakeHOA_status";
         L     0;
         <I;
         JC    storebrakehoaZERO;
         CLR;
         L     "brakeHOA_status";
         L     2;
         >I;
         JC    storebrakehoaZERO;
         CLR;
         A     "brakeoff_pb";
         FP    #ONSH4;
         JC    storebrakehoaZERO;
         CLR;
         A     "brakeon_pb";
         FP    #ONSH5;
         JC    storebrakehoaONE;
         CLR;
         A     "brakeauto_pb";
         FP    #ONSH6;
         JC    storebrakehoaTWO;
         JU    Alarmhorn;





   storebrakehoaZERO:L     0;
         T     "brakeHOA_status";
         BE;

   storebrakehoaONE:L     1;
         T     "brakeHOA_status";
         BE;

   storebrakehoaTWO:L     2;
         T     "brakeHOA_status";
         BE;



   Alarmhorn:L     "alarmhornHOA_status";
         L     0;
         <I;
         JC    storeAlarmhornhoaZERO;
         CLR;
         L     "alarmhornHOA_status";
         L     2;
         >I;
         JC    storeAlarmhornhoaZERO;
         CLR;
         A     "alarmhornoff_pb";
         FP    #ONSH7;
         JC    storeAlarmhornhoaZERO;
         CLR;
         A     "alarmhornon_pb";
         FP    #ONSH8;
         JC    storeAlarmhornhoaONE;
         CLR;
         A     "alarmhornauto_pb";
         FP    #ONSH9;
         JC    storeAlarmhornhoaTWO;
         JU    stationinterlock;





   storeAlarmhornhoaZERO:L     0;
         T     "alarmhornHOA_status";
         BE;

   storeAlarmhornhoaONE:L     1;
         T     "alarmhornHOA_status";
         BE;

   storeAlarmhornhoaTWO:L     2;
         T     "alarmhornHOA_status";
         BE;



   stationinterlock:L     "stationinterlockHOA_status";
         L     0;
         <I;
         JC    storestationinterlockhoaZERO;
         CLR;
         L     "stationinterlockHOA_status";
         L     2;
         >I;
         JC    storestationinterlockhoaZERO;
         CLR;
         A     "stationinterlockoff_pb";
         FP    #ONSH10;
         JC    storestationinterlockhoaZERO;
         CLR;
         A     "stationinterlockon_pb";
         FP    #ONSH11;
         JC    storestationinterlockhoaONE;
         CLR;
         A     "oilpumpVFDauto_pb";
         FP    #ONSH12;
         JC    storestationinterlockhoaTWO;
         JU    endofline;





   storestationinterlockhoaZERO:L     0;
         T     "stationinterlockHOA_status";
         BE;

   storestationinterlockhoaONE:L     1;
         T     "stationinterlockHOA_status";
         BE;

   storestationinterlockhoaTWO:L     2;
         T     "stationinterlockHOA_status";
         BE;

   endofline:BE;
END_REGION
END_FUNCTION_BLOCK

FUNCTION_BLOCK "ALARM_LAD"   // FB10, LAD
{ S7_Optimized_Access := 'TRUE' }
VERSION : 0.1
   VAR
      oillowflowdelayvalue : Int;
      oillowflowdelay : Time;
      ONSA1 : Bool;
      overcuurentdelayvalue : Int;
      overcurrentdelay : Time;
      ONSA2 : Bool;
      oilhightempdelay : Time;
      ONSA3 : Bool;
      rotoroverspeeddelayvalue : Int;
      rotoroverspeeddelay : Time;
      ONSA4 : Bool;
      oilhighflowdelayvalue : Int;
      ONSA5 : Bool;
      brakefailuredelayvalue : Int;
      brakefailuredelay : Time;
      ONSA6 : Bool;
      ONSA7 : Bool;
      oilhightempdelayvalue : Int;
      onsa8 : Bool;
   END_VAR
   VAR_TEMP
      oilhighflowdelay : Time;
      alarmhorntrigger : Bool;
   END_VAR
   VAR_TEMP   // added for the SCL form of the ladder/FBD networks
      _w1 : Bool;
      _w2 : Bool;
   END_VAR
BEGIN

REGION Network 1
   // oillowflowalarm
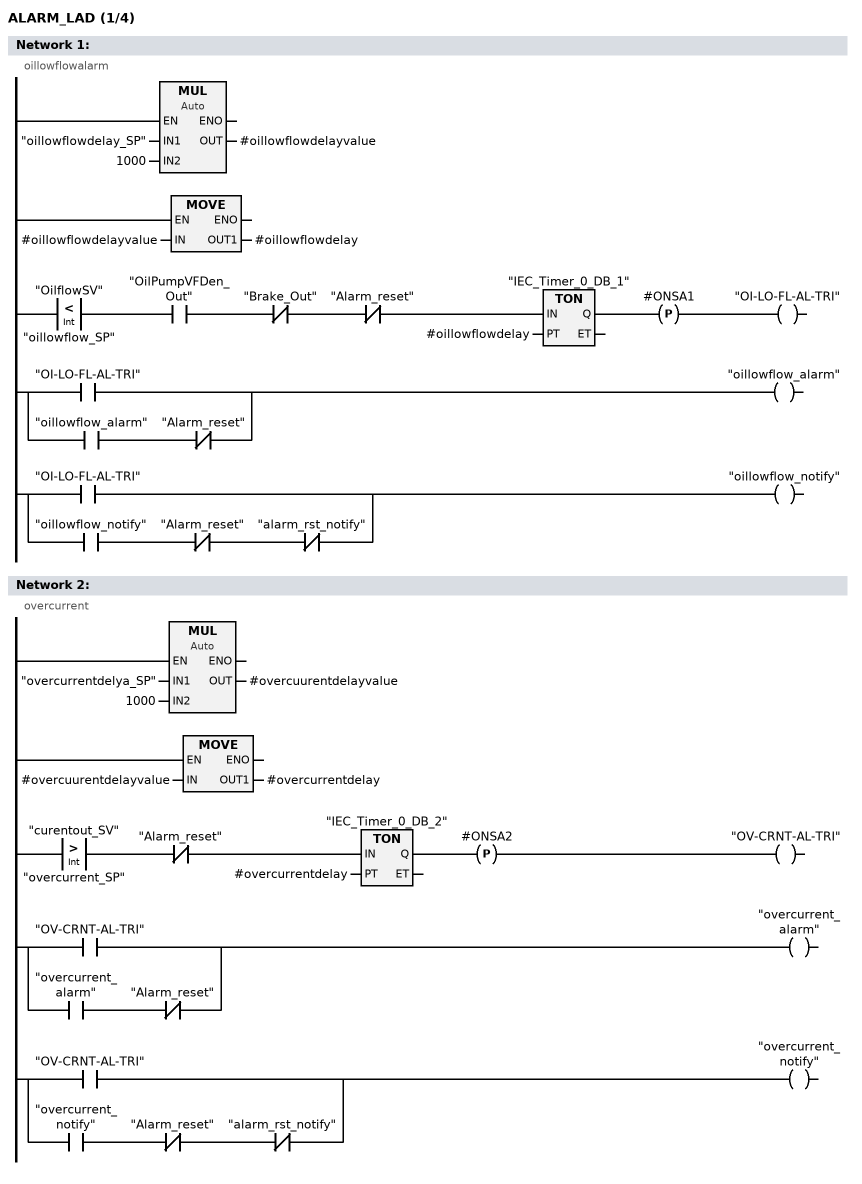
   #oillowflowdelayvalue := "oillowflowdelay_SP" * 1000;
   #oillowflowdelay := #oillowflowdelayvalue;
   "IEC_Timer_0_DB_1".TON(IN := ("OilflowSV" < "oillowflow_SP") AND "OilPumpVFDen_Out" AND NOT "Brake_Out" AND NOT "Alarm_reset",
                          PT := #oillowflowdelay);
   #_w1 := "IEC_Timer_0_DB_1".Q AND NOT #ONSA1;   // rising edge
   #ONSA1 := "IEC_Timer_0_DB_1".Q;
   "OI-LO-FL-AL-TRI" := #_w1;
   "oillowflow_alarm" := "OI-LO-FL-AL-TRI" OR ("oillowflow_alarm" AND NOT "Alarm_reset");
   "oillowflow_notify" := "OI-LO-FL-AL-TRI" OR ("oillowflow_notify" AND NOT "Alarm_reset" AND NOT "alarm_rst_notify");
END_REGION

REGION Network 2
   // overcurrent
   #overcuurentdelayvalue := "overcurrentdelya_SP" * 1000;
   #overcurrentdelay := #overcuurentdelayvalue;
   "IEC_Timer_0_DB_2".TON(IN := ("curentout_SV" > "overcurrent_SP") AND NOT "Alarm_reset",
                          PT := #overcurrentdelay);
   #_w1 := "IEC_Timer_0_DB_2".Q AND NOT #ONSA2;   // rising edge
   #ONSA2 := "IEC_Timer_0_DB_2".Q;
   "OV-CRNT-AL-TRI" := #_w1;
   "overcurrent_alarm" := "OV-CRNT-AL-TRI" OR ("overcurrent_alarm" AND NOT "Alarm_reset");
   "overcurrent_notify" := "OV-CRNT-AL-TRI" OR ("overcurrent_notify" AND NOT "Alarm_reset" AND NOT "alarm_rst_notify");
END_REGION

REGION Network 3
   // Highoiltemp
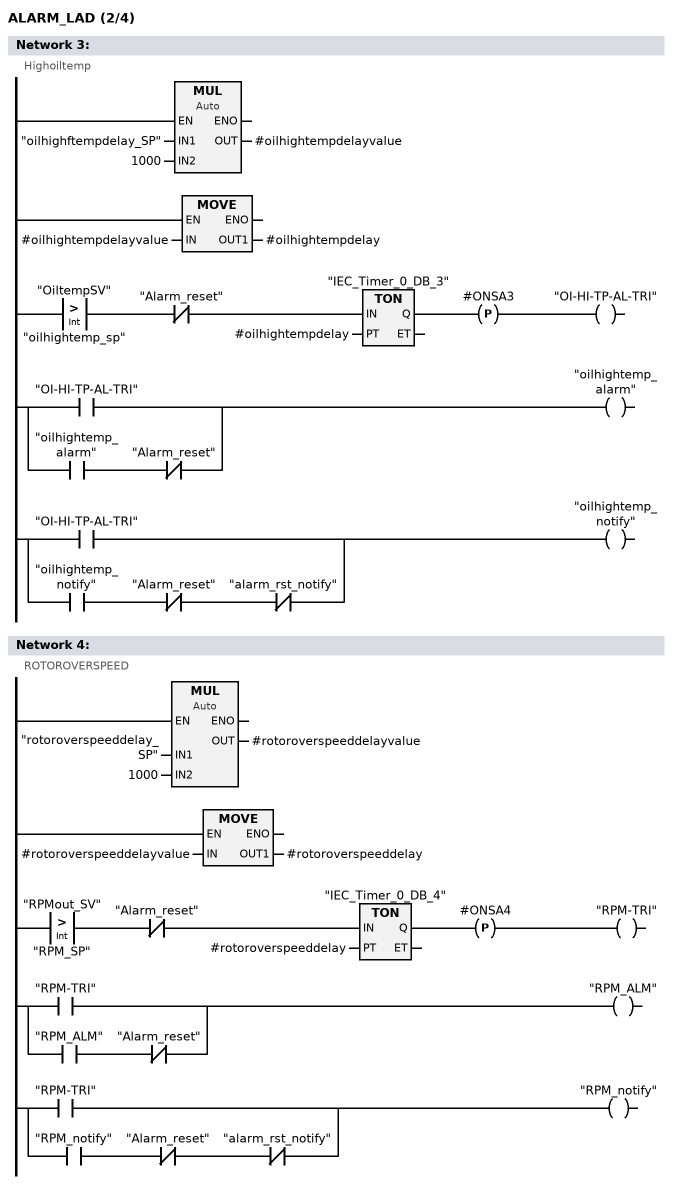
   #oilhightempdelayvalue := "oilhighftempdelay_SP" * 1000;
   #oilhightempdelay := #oilhightempdelayvalue;
   "IEC_Timer_0_DB_3".TON(IN := ("OiltempSV" > "oilhightemp_sp") AND NOT "Alarm_reset", PT := #oilhightempdelay);
   #_w1 := "IEC_Timer_0_DB_3".Q AND NOT #ONSA3;   // rising edge
   #ONSA3 := "IEC_Timer_0_DB_3".Q;
   "OI-HI-TP-AL-TRI" := #_w1;
   "oilhightemp_alarm" := "OI-HI-TP-AL-TRI" OR ("oilhightemp_alarm" AND NOT "Alarm_reset");
   "oilhightemp_notify" := "OI-HI-TP-AL-TRI" OR ("oilhightemp_notify" AND NOT "Alarm_reset" AND NOT "alarm_rst_notify");
END_REGION

REGION Network 4
   // ROTOROVERSPEED
   #rotoroverspeeddelayvalue := "rotoroverspeeddelay_SP" * 1000;
   #rotoroverspeeddelay := #rotoroverspeeddelayvalue;
   "IEC_Timer_0_DB_4".TON(IN := ("RPMout_SV" > "RPM_SP") AND NOT "Alarm_reset", PT := #rotoroverspeeddelay);
   #_w1 := "IEC_Timer_0_DB_4".Q AND NOT #ONSA4;   // rising edge
   #ONSA4 := "IEC_Timer_0_DB_4".Q;
   "RPM-TRI" := #_w1;
   "RPM_ALM" := "RPM-TRI" OR ("RPM_ALM" AND NOT "Alarm_reset");
   "RPM_notify" := "RPM-TRI" OR ("RPM_notify" AND NOT "Alarm_reset" AND NOT "alarm_rst_notify");
END_REGION

REGION Network 5
   // OILHIGHFLOW
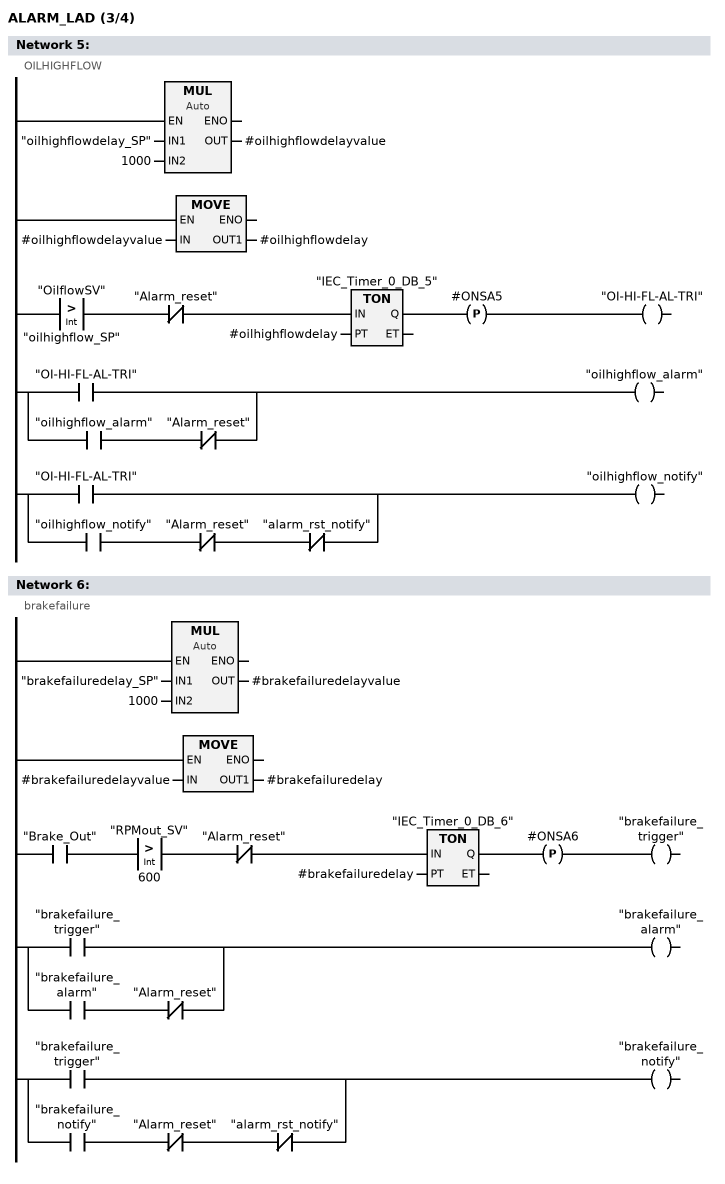
   #oilhighflowdelayvalue := "oilhighflowdelay_SP" * 1000;
   #oilhighflowdelay := #oilhighflowdelayvalue;
   "IEC_Timer_0_DB_5".TON(IN := ("OilflowSV" > "oilhighflow_SP") AND NOT "Alarm_reset", PT := #oilhighflowdelay);
   #_w1 := "IEC_Timer_0_DB_5".Q AND NOT #ONSA5;   // rising edge
   #ONSA5 := "IEC_Timer_0_DB_5".Q;
   "OI-HI-FL-AL-TRI" := #_w1;
   "oilhighflow_alarm" := "OI-HI-FL-AL-TRI" OR ("oilhighflow_alarm" AND NOT "Alarm_reset");
   "oilhighflow_notify" := "OI-HI-FL-AL-TRI" OR ("oilhighflow_notify" AND NOT "Alarm_reset" AND NOT "alarm_rst_notify");
END_REGION

REGION Network 6
   // brakefailure
   #brakefailuredelayvalue := "brakefailuredelay_SP" * 1000;
   #brakefailuredelay := #brakefailuredelayvalue;
   "IEC_Timer_0_DB_6".TON(IN := "Brake_Out" AND ("RPMout_SV" > 600) AND NOT "Alarm_reset",
                          PT := #brakefailuredelay);
   #_w1 := "IEC_Timer_0_DB_6".Q AND NOT #ONSA6;   // rising edge
   #ONSA6 := "IEC_Timer_0_DB_6".Q;
   "brakefailure_trigger" := #_w1;
   "brakefailure_alarm" := "brakefailure_trigger" OR ("brakefailure_alarm" AND NOT "Alarm_reset");
   "brakefailure_notify" := "brakefailure_trigger" OR ("brakefailure_notify" AND NOT "Alarm_reset" AND NOT "alarm_rst_notify");
END_REGION

REGION Network 7
   // E-STOP
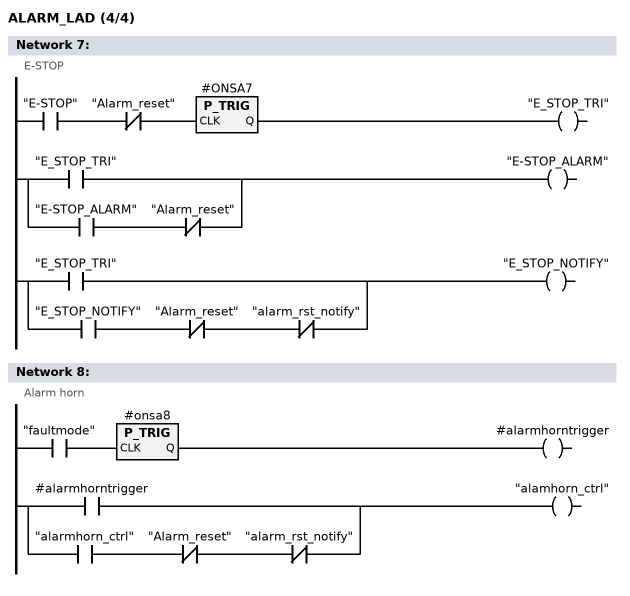
   RUNG wire#powerrail
      Contact( "E-STOP" )
      I_Contact( "Alarm_reset" )
      P_Trig( #ONSA7 )
      Coil( "E_STOP_TRI" )
   END_RUNG
   RUNG wire#powerrail
      Contact( "E_STOP_TRI" )
      wire#w1
      Coil( "E-STOP_ALARM" )
   END_RUNG
   RUNG wire#powerrail
      Contact( "E-STOP_ALARM" )
      I_Contact( "Alarm_reset" )
   END_RUNG wire#w1
   RUNG wire#powerrail
      Contact( "E_STOP_TRI" )
      wire#w2
      Coil( "E_STOP_NOTIFY" )
   END_RUNG
   RUNG wire#powerrail
      Contact( "E_STOP_NOTIFY" )
      I_Contact( "Alarm_reset" )
      I_Contact( "alarm_rst_notify" )
   END_RUNG wire#w2
   // the same network as SCL:
   #_w1 := "E-STOP" AND NOT "Alarm_reset";
   #_w2 := #_w1 AND NOT #ONSA7;   // rising edge
   #ONSA7 := #_w1;
   "E_STOP_TRI" := #_w2;
   "E-STOP_ALARM" := "E_STOP_TRI" OR ("E-STOP_ALARM" AND NOT "Alarm_reset");
   "E_STOP_NOTIFY" := "E_STOP_TRI" OR ("E_STOP_NOTIFY" AND NOT "Alarm_reset" AND NOT "alarm_rst_notify");
END_REGION

REGION Network 8
   // Alarm horn
   RUNG wire#powerrail
      Contact( "faultmode" )
      P_Trig( #onsa8 )
      Coil( #alarmhorntrigger )
   END_RUNG
   RUNG wire#powerrail
      Contact( #alarmhorntrigger )
      wire#w1
      Coil( "alamhorn_ctrl" )
   END_RUNG
   RUNG wire#powerrail
      Contact( "alarmhorn_ctrl" )
      I_Contact( "Alarm_reset" )
      I_Contact( "alarm_rst_notify" )
   END_RUNG wire#w1
   // the same network as SCL:
   #_w1 := "faultmode" AND NOT #onsa8;   // rising edge
   #onsa8 := "faultmode";
   #alarmhorntrigger := #_w1;
   "alamhorn_ctrl" := #alarmhorntrigger OR ("alarmhorn_ctrl" AND NOT "Alarm_reset" AND NOT "alarm_rst_notify");
END_REGION
END_FUNCTION_BLOCK

FUNCTION_BLOCK "ALARM_FBD"   // FB11, FBD
{ S7_Optimized_Access := 'TRUE' }
VERSION : 0.1
   VAR
      ONSA1 : Bool;
      ONSA2 : Bool;
      ONSA3 : Bool;
      ONSA4 : Bool;
      ONSA5 : Bool;
      ONSA6 : Bool;
      ONSA7 : Bool;
      onsa8 : Bool;
   END_VAR
   VAR_TEMP
      ttv1 : Int;
      tt1 : Time;
      ttv2 : Int;
      tt2 : Time;
      ttv3 : Int;
      tt3 : Time;
      ttv4 : Int;
      tt4 : Time;
      ttv5 : Int;
      tt5 : Time;
      ttv6 : Int;
      tt6 : Time;
      alarmtrigger : Bool;
   END_VAR
   VAR_TEMP   // added for the SCL form of the ladder/FBD networks
      _w1 : Bool;
      _w2 : Bool;
   END_VAR
BEGIN

REGION Network 1
   // oillowflowalarm
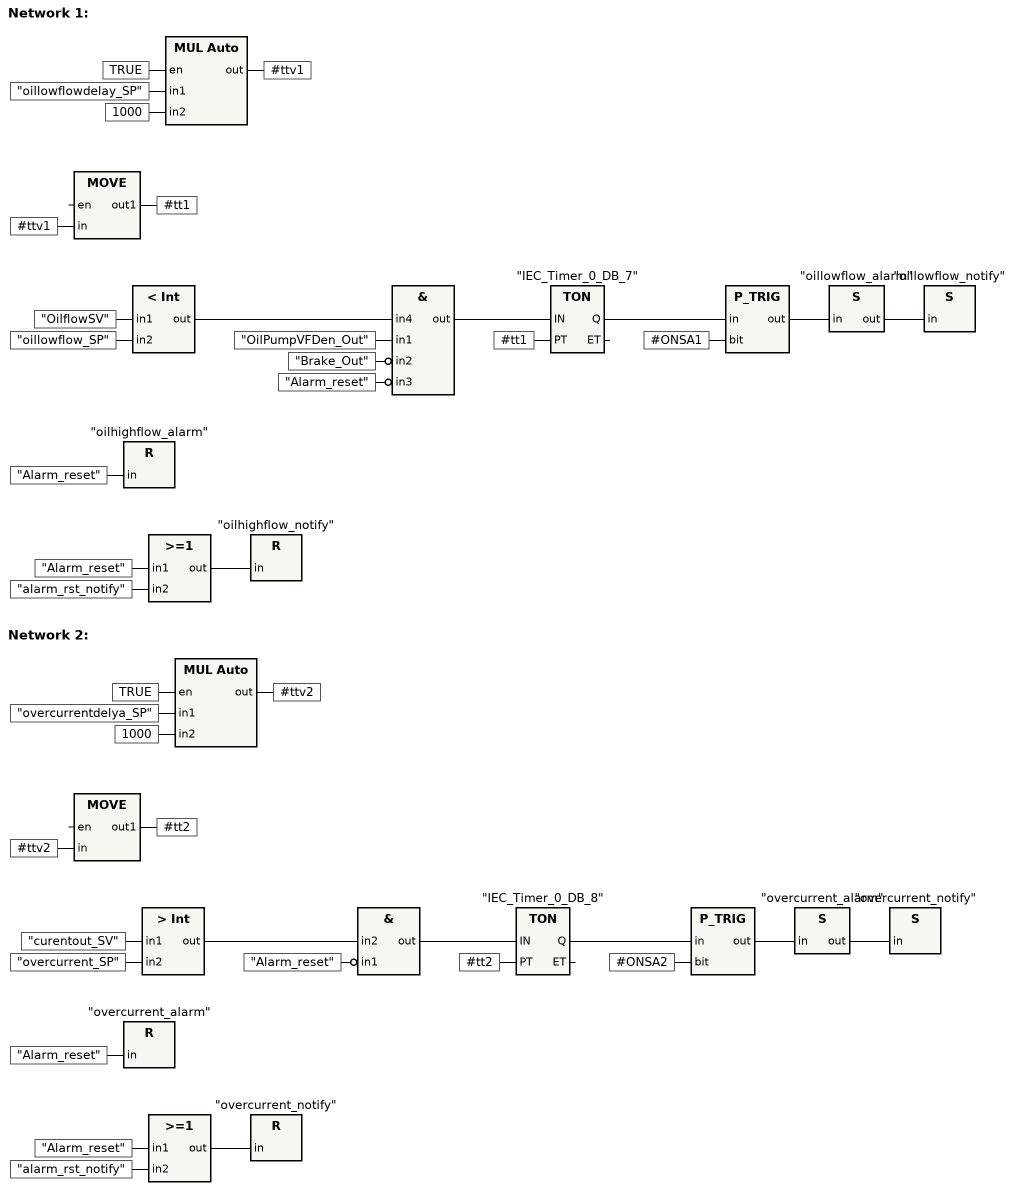
   IF TRUE THEN #ttv1 := "oillowflowdelay_SP" * 1000; END_IF;
   #tt1 := #ttv1;
   "IEC_Timer_0_DB_7".TON(IN := ("OilflowSV" < "oillowflow_SP") AND "OilPumpVFDen_Out" AND NOT "Brake_Out" AND NOT "Alarm_reset",
                          PT := #tt1);
   #_w1 := "IEC_Timer_0_DB_7".Q AND NOT #ONSA1;   // rising edge
   #ONSA1 := "IEC_Timer_0_DB_7".Q;
   IF #_w1 THEN
       "oillowflow_alarm" := TRUE;
       "oillowflow_notify" := TRUE;
   END_IF;
   IF "Alarm_reset" THEN "oilhighflow_alarm" := FALSE; END_IF;
   IF "Alarm_reset" OR "alarm_rst_notify" THEN "oilhighflow_notify" := FALSE; END_IF;
END_REGION

REGION Network 2
   // overcurrent
   IF TRUE THEN #ttv2 := "overcurrentdelya_SP" * 1000; END_IF;
   #tt2 := #ttv2;
   "IEC_Timer_0_DB_8".TON(IN := ("curentout_SV" > "overcurrent_SP") AND NOT "Alarm_reset", PT := #tt2);
   #_w1 := "IEC_Timer_0_DB_8".Q AND NOT #ONSA2;   // rising edge
   #ONSA2 := "IEC_Timer_0_DB_8".Q;
   IF #_w1 THEN
       "overcurrent_alarm" := TRUE;
       "overcurrent_notify" := TRUE;
   END_IF;
   IF "Alarm_reset" THEN "overcurrent_alarm" := FALSE; END_IF;
   IF "Alarm_reset" OR "alarm_rst_notify" THEN "overcurrent_notify" := FALSE; END_IF;
END_REGION

REGION Network 3
   // Highoilflow
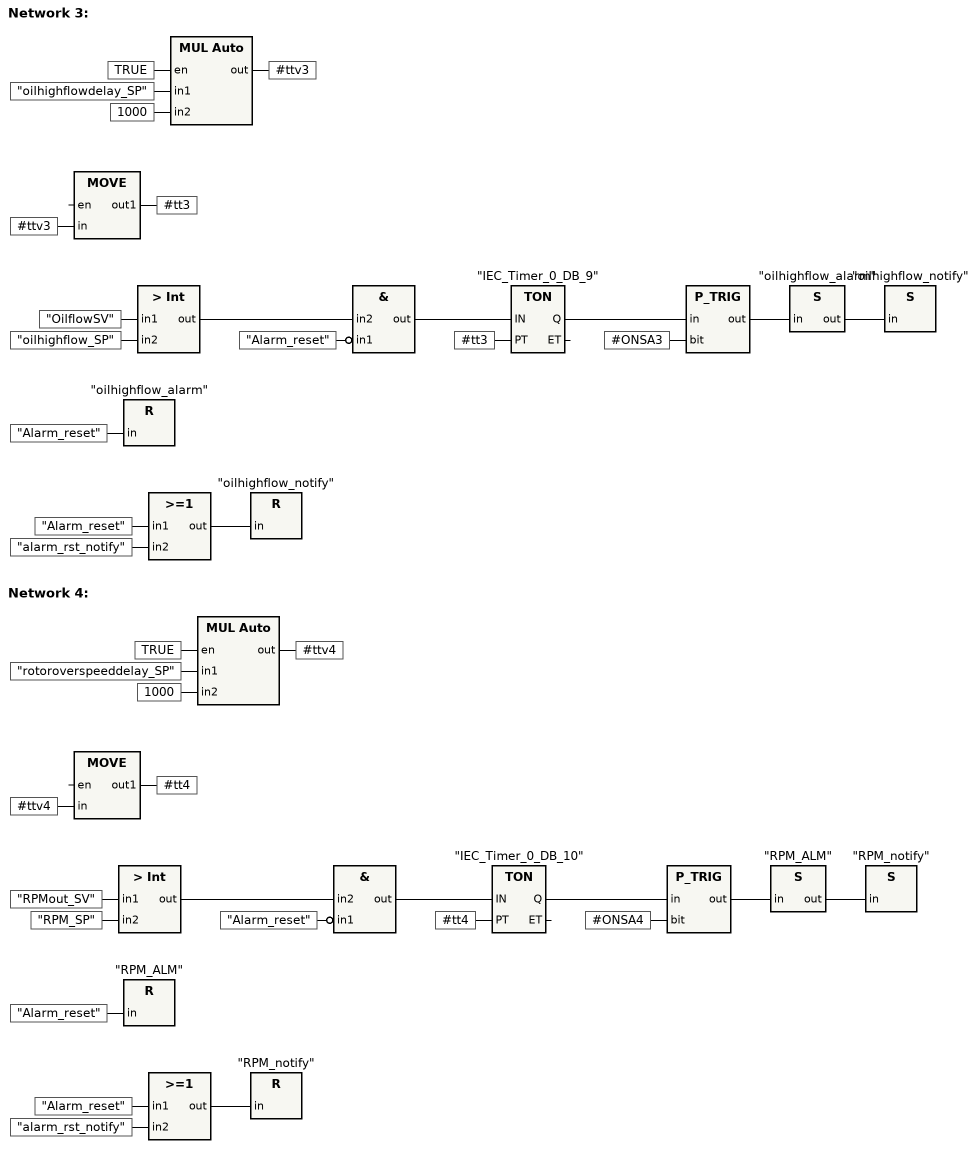
   IF TRUE THEN #ttv3 := "oilhighflowdelay_SP" * 1000; END_IF;
   #tt3 := #ttv3;
   "IEC_Timer_0_DB_9".TON(IN := ("OilflowSV" > "oilhighflow_SP") AND NOT "Alarm_reset", PT := #tt3);
   #_w1 := "IEC_Timer_0_DB_9".Q AND NOT #ONSA3;   // rising edge
   #ONSA3 := "IEC_Timer_0_DB_9".Q;
   IF #_w1 THEN
       "oilhighflow_alarm" := TRUE;
       "oilhighflow_notify" := TRUE;
   END_IF;
   IF "Alarm_reset" THEN "oilhighflow_alarm" := FALSE; END_IF;
   IF "Alarm_reset" OR "alarm_rst_notify" THEN "oilhighflow_notify" := FALSE; END_IF;
END_REGION

REGION Network 4
   // RPM
   IF TRUE THEN #ttv4 := "rotoroverspeeddelay_SP" * 1000; END_IF;
   #tt4 := #ttv4;
   "IEC_Timer_0_DB_10".TON(IN := ("RPMout_SV" > "RPM_SP") AND NOT "Alarm_reset", PT := #tt4);
   #_w1 := "IEC_Timer_0_DB_10".Q AND NOT #ONSA4;   // rising edge
   #ONSA4 := "IEC_Timer_0_DB_10".Q;
   IF #_w1 THEN
       "RPM_ALM" := TRUE;
       "RPM_notify" := TRUE;
   END_IF;
   IF "Alarm_reset" THEN "RPM_ALM" := FALSE; END_IF;
   IF "Alarm_reset" OR "alarm_rst_notify" THEN "RPM_notify" := FALSE; END_IF;
END_REGION

REGION Network 5
   // oilhightemp
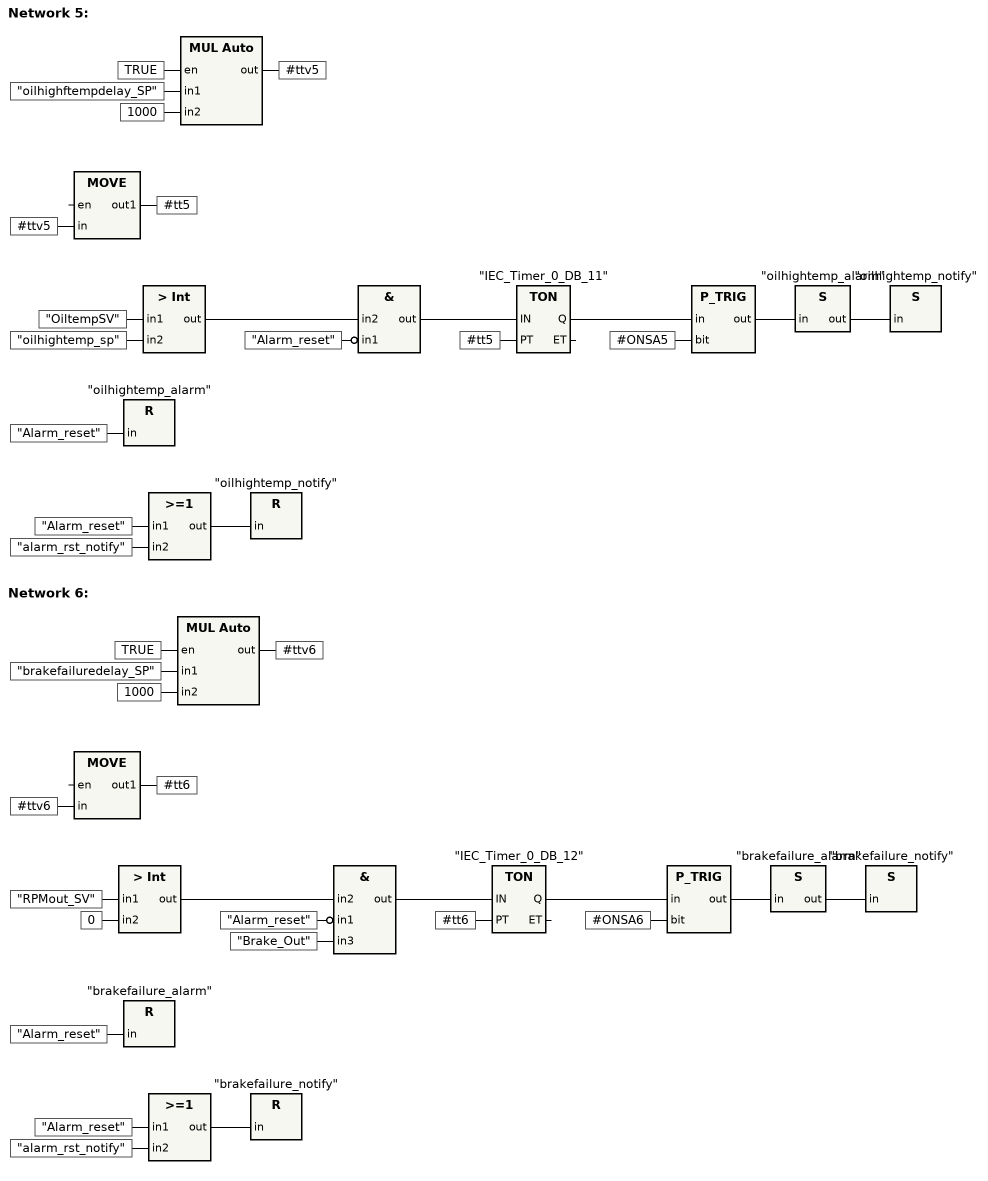
   IF TRUE THEN #ttv5 := "oilhighftempdelay_SP" * 1000; END_IF;
   #tt5 := #ttv5;
   "IEC_Timer_0_DB_11".TON(IN := ("OiltempSV" > "oilhightemp_sp") AND NOT "Alarm_reset", PT := #tt5);
   #_w1 := "IEC_Timer_0_DB_11".Q AND NOT #ONSA5;   // rising edge
   #ONSA5 := "IEC_Timer_0_DB_11".Q;
   IF #_w1 THEN
       "oilhightemp_alarm" := TRUE;
       "oilhightemp_notify" := TRUE;
   END_IF;
   IF "Alarm_reset" THEN "oilhightemp_alarm" := FALSE; END_IF;
   IF "Alarm_reset" OR "alarm_rst_notify" THEN "oilhightemp_notify" := FALSE; END_IF;
END_REGION

REGION Network 6
   // brakefailure
   IF TRUE THEN #ttv6 := "brakefailuredelay_SP" * 1000; END_IF;
   #tt6 := #ttv6;
   "IEC_Timer_0_DB_12".TON(IN := ("RPMout_SV" > 0) AND NOT "Alarm_reset" AND "Brake_Out", PT := #tt6);
   #_w1 := "IEC_Timer_0_DB_12".Q AND NOT #ONSA6;   // rising edge
   #ONSA6 := "IEC_Timer_0_DB_12".Q;
   IF #_w1 THEN
       "brakefailure_alarm" := TRUE;
       "brakefailure_notify" := TRUE;
   END_IF;
   IF "Alarm_reset" THEN "brakefailure_alarm" := FALSE; END_IF;
   IF "Alarm_reset" OR "alarm_rst_notify" THEN "brakefailure_notify" := FALSE; END_IF;
END_REGION

REGION Network 7
   // E-stop
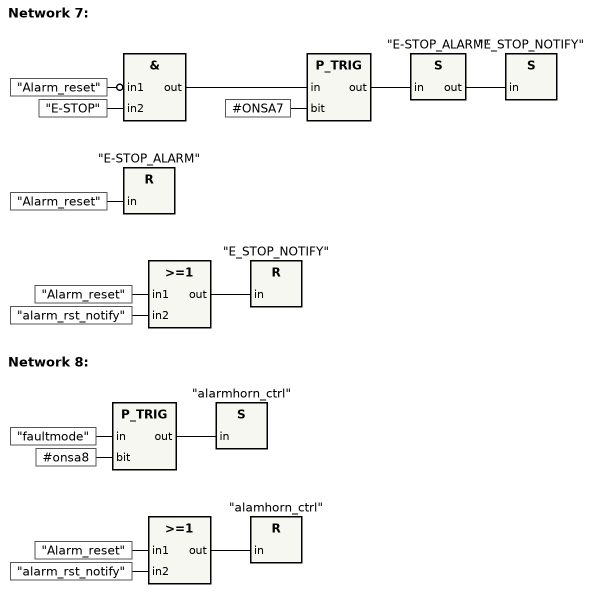
   #_w1 := NOT "Alarm_reset" AND "E-STOP";
   #_w2 := #_w1 AND NOT #ONSA7;   // rising edge
   #ONSA7 := #_w1;
   IF #_w2 THEN
       "E-STOP_ALARM" := TRUE;
       "E_STOP_NOTIFY" := TRUE;
   END_IF;
   IF "Alarm_reset" THEN "E-STOP_ALARM" := FALSE; END_IF;
   IF "Alarm_reset" OR "alarm_rst_notify" THEN "E_STOP_NOTIFY" := FALSE; END_IF;
END_REGION

REGION Network 8
   #_w1 := "faultmode" AND NOT #onsa8;   // rising edge
   #onsa8 := "faultmode";
   IF #_w1 THEN "alarmhorn_ctrl" := TRUE; END_IF;
   IF "Alarm_reset" OR "alarm_rst_notify" THEN "alamhorn_ctrl" := FALSE; END_IF;
END_REGION
END_FUNCTION_BLOCK

FUNCTION_BLOCK "ALARM_SCL"   // FB12, SCL
{ S7_Optimized_Access := 'TRUE' }
VERSION : 0.1
   VAR_TEMP
      tt1 : Time;
      t1 : Time;
      tt2 : Time;
      t2 : Time;
      tt3 : Time;
      t3 : Time;
      tt4 : Time;
      t4 : Time;
      tt5 : Time;
      t5 : Time;
      tt6 : Time;
      t6 : Time;
   END_VAR
BEGIN
   // oillowflow

   IF "OilflowSV" < "oillowflow_SP" AND "OilPumpVFDen_Out" AND NOT "Brake_Out" AND NOT "Alarm_reset" AND NOT "oillowflow_alarm" THEN
       "CONVERTTIME"(VALUEIN := "oillowflowdelay_SP",
                     Time1 => #tt1);

       "IEC_Timer_0_DB_14".TON(IN := TRUE,
                               PT := #tt1,
                               Q => "OI-LO-FL-AL-TRI",
                               ET => #t1);
   ELSE
       RESET_TIMER("IEC_Timer_0_DB_14");

   END_IF;

   IF "OI-LO-FL-AL-TRI" THEN
       "oillowflow_alarm" := 1;
       "oillowflow_notify" := 1;
   END_IF;

   IF "Alarm_reset" AND "oillowflow_alarm"  THEN
       "oillowflow_alarm" := 0;
       "oillowflow_notify" := 0;
   END_IF;

   IF "alarm_rst_notify" AND "oillowflow_notify" THEN
       "oillowflow_notify" := 0;
   END_IF;



   // overcurrent

   IF "curentout_SV" > "overcurrent_SP"  AND NOT "Alarm_reset" AND NOT "overcurrent_alarm" THEN
       "CONVERTTIME"(VALUEIN := "overcurrentdelya_SP",
                     Time1 => #tt2);

       "IEC_Timer_0_DB_15".TON(IN := TRUE,
                               PT := #tt2,
                               Q => "OV-CRNT-AL-TRI",
                               ET => #t2);
   ELSE
       RESET_TIMER("IEC_Timer_0_DB_15");
   END_IF;


   IF "OV-CRNT-AL-TRI" THEN
       "overcurrent_alarm" := 1;
       "overcurrent_notify" := 1;
   END_IF;

   IF "Alarm_reset" AND "overcurrent_alarm" THEN
       "overcurrent_alarm" := 0;
       "overcurrent_notify" := 0;
   END_IF;

   IF "alarm_rst_notify" AND  "overcurrent_notify" THEN
       "overcurrent_notify" := 0;
   END_IF;


   // highoiltemp

   IF "OiltempSV" > "oilhightemp_sp" AND NOT "Alarm_reset" AND NOT "oilhightemp_alarm" THEN
       "CONVERTTIME"(VALUEIN := "oilhighftempdelay_SP",
                     Time1 => #tt3);
       "IEC_Timer_0_DB_16".TON(IN := TRUE,
                               PT := #tt3,
                               Q => "OI-HI-TP-AL-TRI",
                               ET => #t3);

   ELSE
       RESET_TIMER("IEC_Timer_0_DB_16");

   END_IF;

   IF "OI-HI-TP-AL-TRI" THEN
       "oilhightemp_alarm" := 1;
       "oilhightemp_notify" := 1;
   END_IF;

   IF "Alarm_reset" AND "oilhightemp_alarm" THEN
       "oilhightemp_alarm" := 0;
       "oilhightemp_notify" := 0;
   END_IF;

   IF "alarm_rst_notify" AND "oilhightemp_notify" THEN
       "oilhightemp_notify" := 0;
   END_IF;


   // RPM

   IF "RPMout_SV" > "RPM_SP" AND NOT "Alarm_reset" AND NOT "RPM_ALM" THEN
       "CONVERTTIME"(VALUEIN := "rotoroverspeeddelay_SP",
                     Time1 => #tt4);
       "IEC_Timer_0_DB_17".TON(IN := TRUE,
                               PT := #tt4,
                               Q => "RPM-TRI",
                               ET => #t4);
   ELSE

       RESET_TIMER("IEC_Timer_0_DB_17");

   END_IF;

   IF "RPM-TRI" THEN
       "RPM_ALM" := 1;
       "RPM_notify" := 1;
   END_IF;

   IF "Alarm_reset" AND "RPM_ALM" THEN
        "RPM_ALM" := 0;
       "RPM_notify" := 0;
   END_IF;

   IF "alarm_rst_notify" AND  "RPM_notify" THEN
        "RPM_notify" := 0;
   END_IF;


   // OILHIGHFLOW

   IF "OilflowSV" > "oilhighflow_SP" AND NOT "Alarm_reset" AND NOT "oilhighflow_alarm" THEN
       "CONVERTTIME"(VALUEIN := "oilhighflowdelay_SP",
                     Time1 => #tt5);

       "IEC_Timer_0_DB_18".TON(IN := TRUE,
                               PT := #tt5,
                               Q => "OI-HI-FL-AL-TRI",
                               ET => #t5);
   ELSE
       RESET_TIMER("IEC_Timer_0_DB_18");


   END_IF;

   IF "OI-HI-FL-AL-TRI" THEN
       "oilhighflow_alarm" := 1;
       "oilhighflow_notify" := 1;
   END_IF;

   IF "Alarm_reset" AND "oilhighflow_alarm" THEN
       "oilhighflow_alarm" := 0;
       "oilhighflow_notify" := 0;
   END_IF;

   IF "alarm_rst_notify" AND "oilhighflow_notify" THEN
       "oilhighflow_notify" := 0;
   END_IF;


   // BRAKE

   IF "RPMout_SV" < 0 AND "Brake_Out" AND NOT "Alarm_reset" AND NOT "brakefailure_alarm" THEN
       "CONVERTTIME"(VALUEIN := "brakefailuredelay_SP",
                     Time1 => #tt6);

       "IEC_Timer_0_DB_19".TON(IN := TRUE,
                               PT := #tt6,
                               Q => "brakefailure_trigger",
                               ET => #t6);
   ELSE
       RESET_TIMER("IEC_Timer_0_DB_19");

   END_IF;

   IF "brakefailure_trigger" THEN
       "brakefailure_alarm" := 1;
       "brakefailure_notify" := 1;
   END_IF;

   IF "Alarm_reset" AND "brakefailure_alarm"THEN
       "brakefailure_alarm" := 0;
       "brakefailure_notify" := 0;
   END_IF;

   IF "alarm_rst_notify" AND "brakefailure_notify" THEN
       "brakefailure_notify" := 0;
   END_IF;


   // E-STOP

   IF "E-STOP"   AND  NOT "Alarm_reset" AND NOT "E-STOP_ALARM"   THEN


       "E-STOP_ALARM" := 1;
       "E_STOP_NOTIFY" := 1;
   END_IF;

   IF "Alarm_reset" AND  "E-STOP_ALARM" THEN
       "E-STOP_ALARM" := 0;
       "E_STOP_NOTIFY" := 0;
   END_IF;

   IF "alarm_rst_notify" AND "E_STOP_NOTIFY" THEN
       "E_STOP_NOTIFY" := 0;
   END_IF;

   IF "faultmode" AND NOT "alarmhorn_ctrl" THEN
       "alarmhorn_ctrl" := 1;
   ELSE
       "alarmhorn_ctrl" := 0;
   END_IF;

   IF "alarmhorn_ctrl" AND  "Alarm_reset" OR "alarm_rst_notify" THEN
       "alamhorn_ctrl" := 0;
   END_IF;
END_FUNCTION_BLOCK

FUNCTION_BLOCK "ALARM_STL"   // FB13, STL
{ S7_Optimized_Access := 'TRUE' }
VERSION : 0.1
   VAR
      OSA1 : Bool;
      OSA2 : Bool;
      OSA3 : Bool;
      OSA4 : Bool;
      OSA5 : Bool;
      OSA6 : Bool;
      OSA7 : Bool;
      OSA8 : Bool;
      OSA9 : Bool;
      OSA10 : Bool;
      OSA11 : Bool;
      OSA12 : Bool;
      OSA13 : Bool;
      OSA14 : Bool;
      OSA15 : Bool;
      osa16 : Bool;
      OSA17 : Bool;
   END_VAR
   VAR_TEMP
      TT1 : Time;
      TT2 : Time;
      TT3 : Time;
      TT4 : Time;
      TT5 : Time;
      TT6 : Time;
      TT7 : Time;
      T1 : Time;
      T2 : Time;
      T3 : Time;
      T4 : Time;
      T5 : Time;
      T6 : Time;
      T7 : Time;
   END_VAR
BEGIN

REGION Network 1
   //oillowflowalarm

         L     "OilflowSV";
         L     "oillowflow_SP";
         <I;
         A     "OilPumpVFDen_Out";
         AN    "Brake_Out";
         AN    "Alarm_reset";
         JC    TIMING;
         CLR;
         A     "Alarm_reset";
         FP    #OSA1;
         JC    ALARMRESET;
         CLR;
         A     "alarm_rst_notify";
         FP    #OSA2;
         JC    ALARMNOTIFYRESET;
         JU    OVERCURRENT;

   TIMING:CALL  "CONVERTTIME"
         ( VALUEIN := "oillowflowdelay_SP",
           Time1   := #TT1
         );

         CALL  TON, "IEC_Timer_0_DB_20"
         ( IN := TRUE,
           PT := #TT1,
           Q  := "OI-LO-FL-AL-TRI",
           ET := #T1
         );
         A     "OI-LO-FL-AL-TRI";
         JC    SETALARM;


         JU    OVERCURRENT;

   SETALARM:S     "oillowflow_alarm";
         S     "oillowflow_notify";
         JU    OVERCURRENT;

   ALARMRESET:R     "oillowflow_alarm";
         R     "oillowflow_notify";
         CALL  RESET_TIMER
         ( "TIMER" := "IEC_Timer_0_DB_20"
         );

         JU    OVERCURRENT;

   ALARMNOTIFYRESET:R     "oillowflow_notify";
         JU    OVERCURRENT;



   //overcurrent

   OVERCURRENT:L     "curentout_SV";
         L     "overcurrent_SP";
         >I;
         AN    "Alarm_reset";
         JC    OCTIMING;
         CLR;
         A     "Alarm_reset";
         FP    #OSA3;
         JC    OCALARMRESET;
         CLR;
         A     "alarm_rst_notify";
         FP    #OSA4;
         JC    OCALARMNOTIFYRESET;

         JU    HIGHOIL;

   OCTIMING:CALL  "CONVERTTIME"
         ( VALUEIN := "overcurrentdelya_SP",
           Time1   := #TT2
         );

         CALL  TON, "IEC_Timer_0_DB_21"
         ( IN := TRUE,
           PT := #TT2,
           Q  := "OV-CRNT-AL-TRI",
           ET := #T2
         );
         A     "OV-CRNT-AL-TRI";
         JC    OCSETALARM;


         JU    HIGHOIL;

   OCSETALARM:S     "overcurrent_alarm";
         S     "overcurrent_notify";
         JU    HIGHOIL;

   OCALARMRESET:R     "overcurrent_alarm";
         R     "overcurrent_notify";
         CALL  RESET_TIMER
         ( "TIMER" := "IEC_Timer_0_DB_21"
         );

         JU    HIGHOIL;

   OCALARMNOTIFYRESET:R     "overcurrent_notify";
         JU    HIGHOIL;




   //Highoiltemp

   HIGHOIL:L     "OiltempSV";
         L     "oilhightemp_sp";
         >I;
         AN    "Alarm_reset";
         JC    hoTIMING;
         CLR;
         A     "Alarm_reset";
         FP    #OSA5;
         JC    hoALARMRESET;
         CLR;
         A     "alarm_rst_notify";
         FP    #OSA6;
         JC    hoALARMNOTIFYRESET;
         JU    OILHIGH;

   hoTIMING:CALL  "CONVERTTIME"
         ( VALUEIN := "oilhighflowdelay_SP",
           Time1   := #TT3
         );

         CALL  TON, "IEC_Timer_0_DB_22"
         ( IN := true,
           PT := #TT3,
           Q  := "OI-HI-TP-AL-TRI",
           ET := #T3
         );
         A     "OI-HI-TP-AL-TRI";
         JC    hoSETALARM;


         JU    OILHIGH;

   hoSETALARM:S     "oilhightemp_alarm";
         S     "oilhightemp_notify";
         JU    OILHIGH;

   hoALARMRESET:R     "oilhightemp_alarm";
         R     "oilhightemp_notify";
         CALL  RESET_TIMER
         ( "TIMER" := "IEC_Timer_0_DB_22"
         );

         JU    OILHIGH;

   hoALARMNOTIFYRESET:R     "oilhightemp_notify";
         JU    OILHIGH;




   //oiLHIGHflowalarm

   OILHIGH:L     "OilflowSV";
         L     "oilhighflow_SP";
         >I;
         AN    "Alarm_reset";
         JC    OHFTIMING;
         CLR;
         A     "Alarm_reset";
         FP    #OSA7;
         JC    OHFALARMRESET;
         CLR;
         A     "alarm_rst_notify";
         FP    #OSA8;
         JC    OHFALARMNOTIFYRESET;
         JU    RPM;

   OHFTIMING:CALL  "CONVERTTIME"
         ( VALUEIN := "oilhighflowdelay_SP",
           Time1   := #TT4
         );
         CALL  TON, "IEC_Timer_0_DB_23"
         ( IN := TRUE,
           PT := #TT4,
           Q  := "OI-HI-FL-AL-TRI",
           ET := #T4
         );
         A     "OI-HI-FL-AL-TRI";

         JC    OHFSETALARM;


         JU    RPM;

   OHFSETALARM:S     "oilhighflow_alarm";
         S     "oilhighflow_notify";
         JU    RPM;

   OHFALARMRESET:R     "oilhighflow_alarm";
         R     "oilhighflow_notify";
         CALL  RESET_TIMER
         ( "TIMER" := "IEC_Timer_0_DB_23"
         );

         JU    RPM;

   OHFALARMNOTIFYRESET:R     "oilhighflow_notify";
         JU    RPM;




   //RPM

   RPM:  L     "RPMout_SV";
         L     "RPM_SP";
         >I;
         AN    "Alarm_reset";
         JC    RPMTIMING;
         CLR;
         A     "Alarm_reset";
         FP    #OSA9;
         JC    RPMALARMRESET;
         CLR;
         A     "alarm_rst_notify";
         FP    #OSA10;
         JC    RPMALARMNOTIFYRESET;
         JU    BRAKEFAILURE;

   RPMTIMING:CALL  "CONVERTTIME"
         ( VALUEIN := "rotoroverspeeddelay_SP",
           Time1   := #TT5
         );

         CALL  TON, "IEC_Timer_0_DB_24"
         ( IN := TRUE,
           PT := #TT5,
           Q  := "RPM-TRI",
           ET := #T5
         );

         A     "RPM-TRI";
         JC    RPMSETALARM;


         JU    BRAKEFAILURE;

   RPMSETALARM:S     "RPM_ALM";
         S     "RPM_notify";
         JU    BRAKEFAILURE;

   RPMALARMRESET:R     "RPM_ALM";
         R     "RPM_notify";
         CALL  RESET_TIMER
         ( "TIMER" := "IEC_Timer_0_DB_24"
         );

         JU    BRAKEFAILURE;

   RPMALARMNOTIFYRESET:R     "RPM_notify";
         JU    BRAKEFAILURE;




   //BRAKEFAILURE

   BRAKEFAILURE:L     "RPMout_SV";
         L     0;
         >I;
         A     "Brake_Out";
         AN    "Alarm_reset";
         JC    BRTIMING;
         CLR;
         A     "Alarm_reset";
         FP    #OSA11;
         JC    BRALARMRESET;
         CLR;
         A     "alarm_rst_notify";
         FP    #OSA2;
         JC    BRALARMNOTIFYRESET;
         JU    ESTOP;

   BRTIMING:CALL  "CONVERTTIME"
         ( VALUEIN := "brakefailuredelay_SP",
           Time1   := #TT6
         );

         CALL  TON, "IEC_Timer_0_DB_26"
         ( IN := TRUE,
           PT := #TT6,
           Q  := "brakefailure_trigger",
           ET := #T5
         );
         A     "brakefailure_trigger";

         JC    BRSETALARM;


         JU    ESTOP;

   BRSETALARM:S     "brakefailure_alarm";
         S     "brakefailure_notify";
         JU    ESTOP;

   BRALARMRESET:R     "brakefailure_alarm";
         R     "brakefailure_notify";
         CALL  RESET_TIMER
         ( "TIMER" := "IEC_Timer_0_DB_26"
         );

         JU    ESTOP;

   BRALARMNOTIFYRESET:R     "brakefailure_notify";
         JU    ESTOP;



   //ESTOP


   ESTOP:A     "E-STOP";
         AN    "Alarm_reset";
         FP    #OSA15;
         JC    ESETALARM;
         CLR;
         A     "Alarm_reset";
         FP    #OSA13;
         JC    EALARMRESET;
         CLR;
         A     "alarm_rst_notify";
         FP    #OSA14;
         JC    EALARMNOTIFYRESET;
         JU    alarmhorn;


   ESETALARM:S     "E-STOP_ALARM";
         S     "E_STOP_NOTIFY";
         JU    alarmhorn;

   EALARMRESET:R     "E-STOP_ALARM";
         R     "E_STOP_NOTIFY";
         JU    alarmhorn;

   EALARMNOTIFYRESET:R     "E_STOP_NOTIFY";
         JU    alarmhorn;



   //alarmhorn


   alarmhorn:A     "faultmode";
         AN    "Alarm_reset";
         FP    #osa16;
         JC    AHSETALARM;
         CLR;
         A     "Alarm_reset";
         O     "alarm_rst_notify";
         FP    #OSA17;
         JC    AHALARMRESET;

         JU    endofline;


   AHSETALARM:S     "alamhorn_ctrl";

         JU    endofline;

   AHALARMRESET:R     "alamhorn_ctrl";

         JU    endofline;


   endofline:BE;
END_REGION
END_FUNCTION_BLOCK

FUNCTION_BLOCK "MODES_LAD"   // FB14, LAD
{ S7_Optimized_Access := 'TRUE' }
VERSION : 0.1
   VAR
      onsa1 : Bool;
      onsa2 : Bool;
      onsa3 : Bool;
      onsa4 : Bool;
      onsa5 : Bool;
      onsa6 : Bool;
   END_VAR
   VAR_TEMP
      TT1 : Time;
      ttt1 : Int;
      ttt2 : Int;
      tt2 : Time;
      Temp_1 : Bool;
      tt3 : Time;
   END_VAR
   VAR_TEMP   // added for the SCL form of the ladder/FBD networks
      _w1 : Bool;
      _w2 : Bool;
      _w3 : Bool;
   END_VAR
BEGIN

REGION Network 1
   // warmupmode
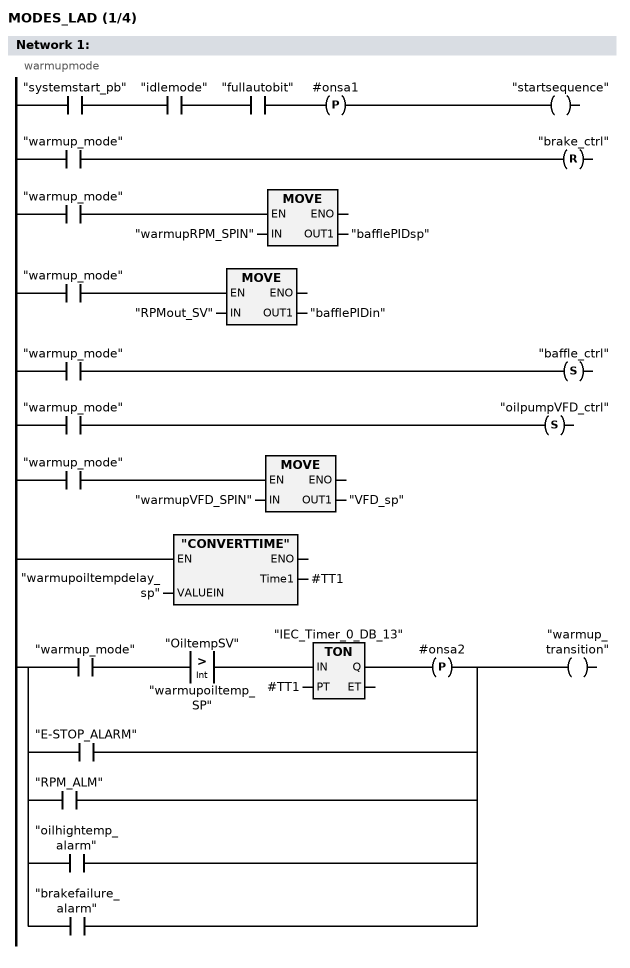
   #_w1 := "systemstart_pb" AND "idlemode" AND "fullautobit";
   #_w2 := #_w1 AND NOT #onsa1;   // rising edge
   #onsa1 := #_w1;
   "startsequence" := #_w2;
   IF "warmup_mode" THEN
       "brake_ctrl" := FALSE;
       "bafflePIDsp" := "warmupRPM_SPIN";
       "bafflePIDin" := "RPMout_SV";
       "baffle_ctrl" := TRUE;
       "oilpumpVFD_ctrl" := TRUE;
       "VFD_sp" := "warmupVFD_SPIN";
   END_IF;
   "CONVERTTIME"(VALUEIN := "warmupoiltempdelay_sp", Time1 => #TT1);
   "IEC_Timer_0_DB_13".TON(IN := "warmup_mode" AND ("OiltempSV" > "warmupoiltemp_SP"), PT := #TT1);
   #_w3 := "IEC_Timer_0_DB_13".Q AND NOT #onsa2;   // rising edge
   #onsa2 := "IEC_Timer_0_DB_13".Q;
   "warmup_transition" := #_w3 OR "E-STOP_ALARM" OR "RPM_ALM" OR "oilhightemp_alarm" OR "brakefailure_alarm";
END_REGION

REGION Network 2
   // stabilize mode
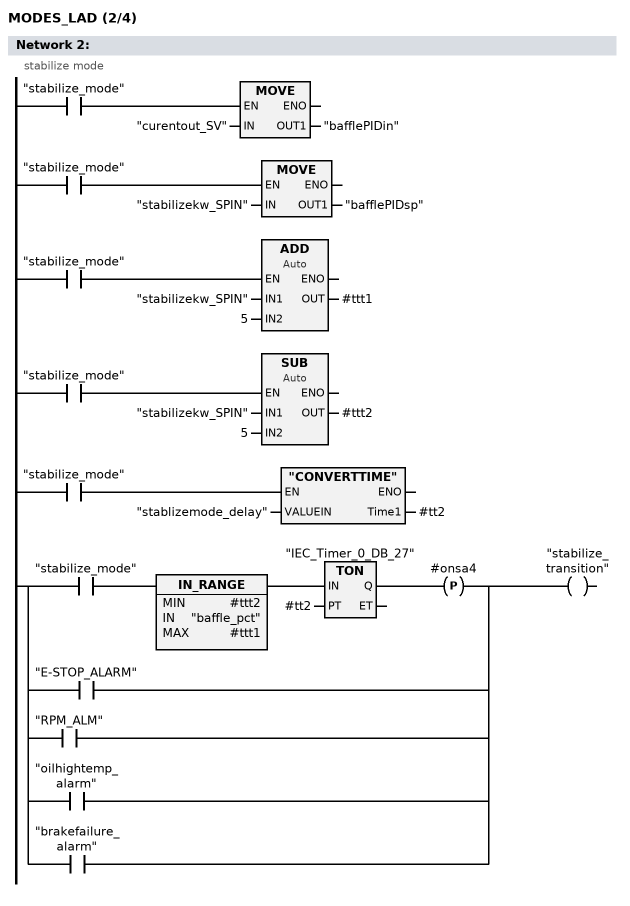
   IF "stabilize_mode" THEN
       "bafflePIDin" := "curentout_SV";
       "bafflePIDsp" := "stabilizekw_SPIN";
       #ttt1 := "stabilizekw_SPIN" + 5;
       #ttt2 := "stabilizekw_SPIN" - 5;
       "CONVERTTIME"(VALUEIN := "stablizemode_delay", Time1 => #tt2);
   END_IF;
   "IEC_Timer_0_DB_27".TON(IN := "stabilize_mode" AND (#ttt2 <= "baffle_pct") AND ("baffle_pct" <= #ttt1),
                           PT := #tt2);
   #_w1 := "IEC_Timer_0_DB_27".Q AND NOT #onsa4;   // rising edge
   #onsa4 := "IEC_Timer_0_DB_27".Q;
   "stabilize_transition" := #_w1 OR "E-STOP_ALARM" OR "RPM_ALM" OR "oilhightemp_alarm" OR "brakefailure_alarm";
END_REGION

REGION Network 3
   // generationmode
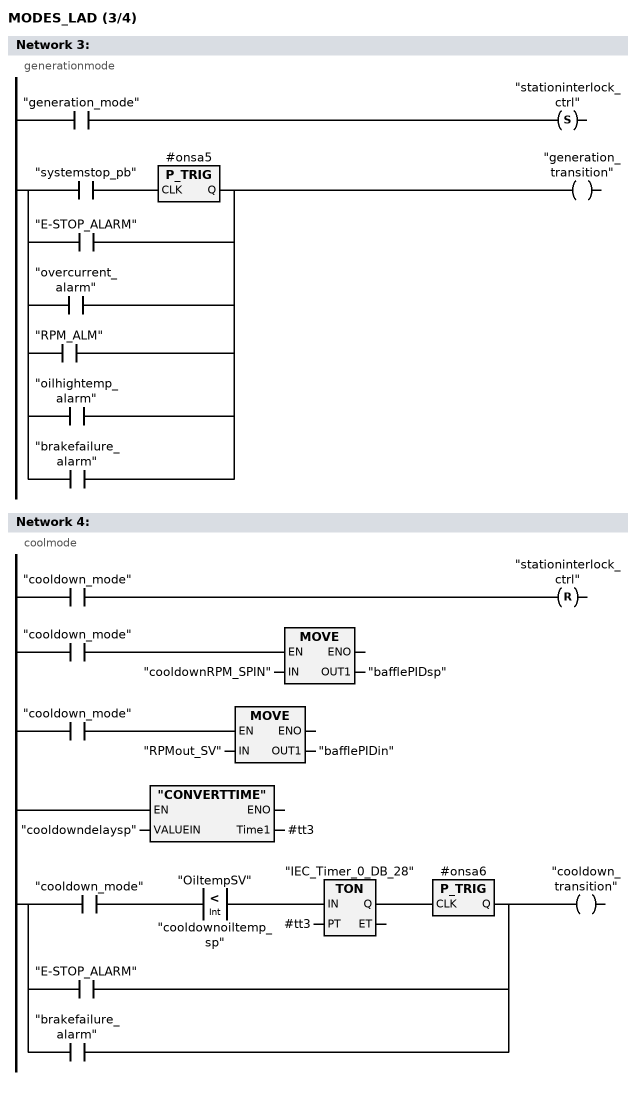
   RUNG wire#powerrail
      Contact( "generation_mode" )
      S_Coil( "stationinterlock_ctrl" )
   END_RUNG
   RUNG wire#powerrail
      Contact( "systemstop_pb" )
      P_Trig( #onsa5 )
      wire#w1
      Coil( "generation_transition" )
   END_RUNG
   RUNG wire#powerrail
      Contact( "E-STOP_ALARM" )
   END_RUNG wire#w1
   RUNG wire#powerrail
      Contact( "overcurrent_alarm" )
   END_RUNG wire#w1
   RUNG wire#powerrail
      Contact( "RPM_ALM" )
   END_RUNG wire#w1
   RUNG wire#powerrail
      Contact( "oilhightemp_alarm" )
   END_RUNG wire#w1
   RUNG wire#powerrail
      Contact( "brakefailure_alarm" )
   END_RUNG wire#w1
   // the same network as SCL:
   IF "generation_mode" THEN "stationinterlock_ctrl" := TRUE; END_IF;
   #_w1 := "systemstop_pb" AND NOT #onsa5;   // rising edge
   #onsa5 := "systemstop_pb";
   "generation_transition" := #_w1 OR "E-STOP_ALARM" OR "overcurrent_alarm" OR "RPM_ALM" OR "oilhightemp_alarm" OR "brakefailure_alarm";
END_REGION

REGION Network 4
   // coolmode
   IF "cooldown_mode" THEN
       "stationinterlock_ctrl" := FALSE;
       "bafflePIDsp" := "cooldownRPM_SPIN";
       "bafflePIDin" := "RPMout_SV";
   END_IF;
   "CONVERTTIME"(VALUEIN := "cooldowndelaysp", Time1 => #tt3);
   "IEC_Timer_0_DB_28".TON(IN := "cooldown_mode" AND ("OiltempSV" < "cooldownoiltemp_sp"), PT := #tt3);
   #_w1 := "IEC_Timer_0_DB_28".Q AND NOT #onsa6;   // rising edge
   #onsa6 := "IEC_Timer_0_DB_28".Q;
   "cooldown_transition" := #_w1 OR "E-STOP_ALARM" OR "brakefailure_alarm";
END_REGION

REGION Network 5
   // idlemode
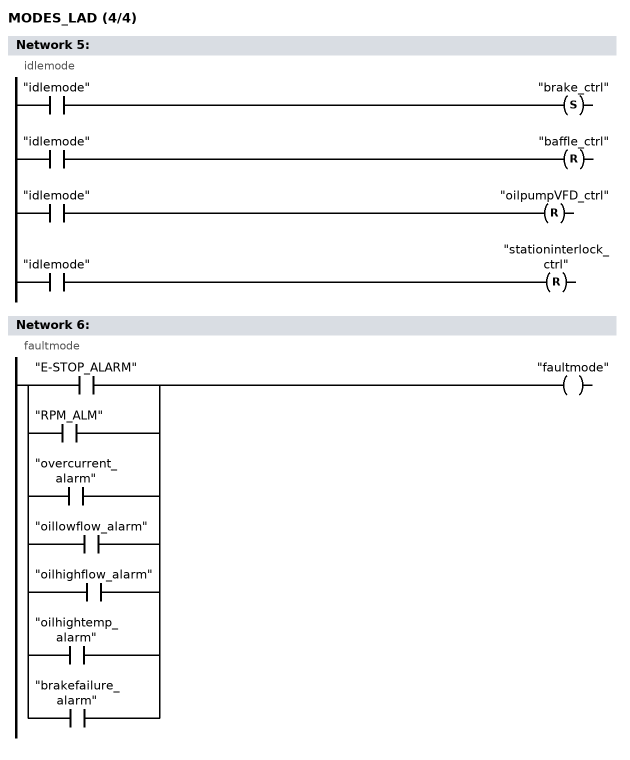
   RUNG wire#powerrail
      Contact( "idlemode" )
      S_Coil( "brake_ctrl" )
   END_RUNG
   RUNG wire#powerrail
      Contact( "idlemode" )
      R_Coil( "baffle_ctrl" )
   END_RUNG
   RUNG wire#powerrail
      Contact( "idlemode" )
      R_Coil( "oilpumpVFD_ctrl" )
   END_RUNG
   RUNG wire#powerrail
      Contact( "idlemode" )
      R_Coil( "stationinterlock_ctrl" )
   END_RUNG
   // the same network as SCL:
   IF "idlemode" THEN
       "brake_ctrl" := TRUE;
       "baffle_ctrl" := FALSE;
       "oilpumpVFD_ctrl" := FALSE;
       "stationinterlock_ctrl" := FALSE;
   END_IF;
END_REGION

REGION Network 6
   // faultmode
   RUNG wire#powerrail
      Contact( "E-STOP_ALARM" )
      wire#w1
      Coil( "faultmode" )
   END_RUNG
   RUNG wire#powerrail
      Contact( "RPM_ALM" )
   END_RUNG wire#w1
   RUNG wire#powerrail
      Contact( "overcurrent_alarm" )
   END_RUNG wire#w1
   RUNG wire#powerrail
      Contact( "oillowflow_alarm" )
   END_RUNG wire#w1
   RUNG wire#powerrail
      Contact( "oilhighflow_alarm" )
   END_RUNG wire#w1
   RUNG wire#powerrail
      Contact( "oilhightemp_alarm" )
   END_RUNG wire#w1
   RUNG wire#powerrail
      Contact( "brakefailure_alarm" )
   END_RUNG wire#w1
   // the same network as SCL:
   "faultmode" := "E-STOP_ALARM" OR "RPM_ALM" OR "overcurrent_alarm" OR "oillowflow_alarm" OR "oilhighflow_alarm" OR "oilhightemp_alarm" OR "brakefailure_alarm";
END_REGION
END_FUNCTION_BLOCK

FUNCTION_BLOCK "MODES_FBD"   // FB15, FBD
{ S7_Optimized_Access := 'TRUE' }
VERSION : 0.1
// – When Start pushbutton is pressed, the sequence begins with this step. Allow the rotor to
// turn at a speed somethere between 20 and 50 RPMs and run the oil pump at some low output level (2-
// 10 GPM maybe?) until the oil temp reaches 150 degrees. Once we’ve maintained at least 150 degrees
// for 10 seconds, we want to transition into the next mode.
// (continued)
// Stabilize – Generator should speed up until desired kW output is attained. Once we’re stable within
// 5kW (+/-) of the setpoint for at least 10 seconds, we should transition into the next mode.
// Generation – Keep everything running and close the interlock.
// Cooldown – Once the Stop button has been pushed, open the interlock, slow the rotor to between 20
// and 50 RPMs and maintain a high oil flow until the oil temp is below 150 degrees. Once we’re below
// for ten seconds, we transition into Idle mode.
// Idle – Interlock and baffle are deenergized and brake is engaged.
// Fault – When we hit an alarm, the sequence should be aborted according to the alarm details (above in
// the Alarms section), and we should go into Fault mode (which is not part of our sequence).
   VAR
      onsa1 : Bool;
      onsa2 : Bool;
      onsa3 : Bool;
      onsa4 : Bool;
      onsa5 : Bool;
   END_VAR
   VAR_TEMP
      tt1 : Time;
      ttt1 : Int;
      ttt2 : Int;
      tt2 : Time;
      tt3 : Time;
   END_VAR
   VAR_TEMP   // added for the SCL form of the ladder/FBD networks
      _w1 : Bool;
      _w2 : Bool;
      _w3 : Bool;
   END_VAR
BEGIN

REGION Network 1
   // startupmode
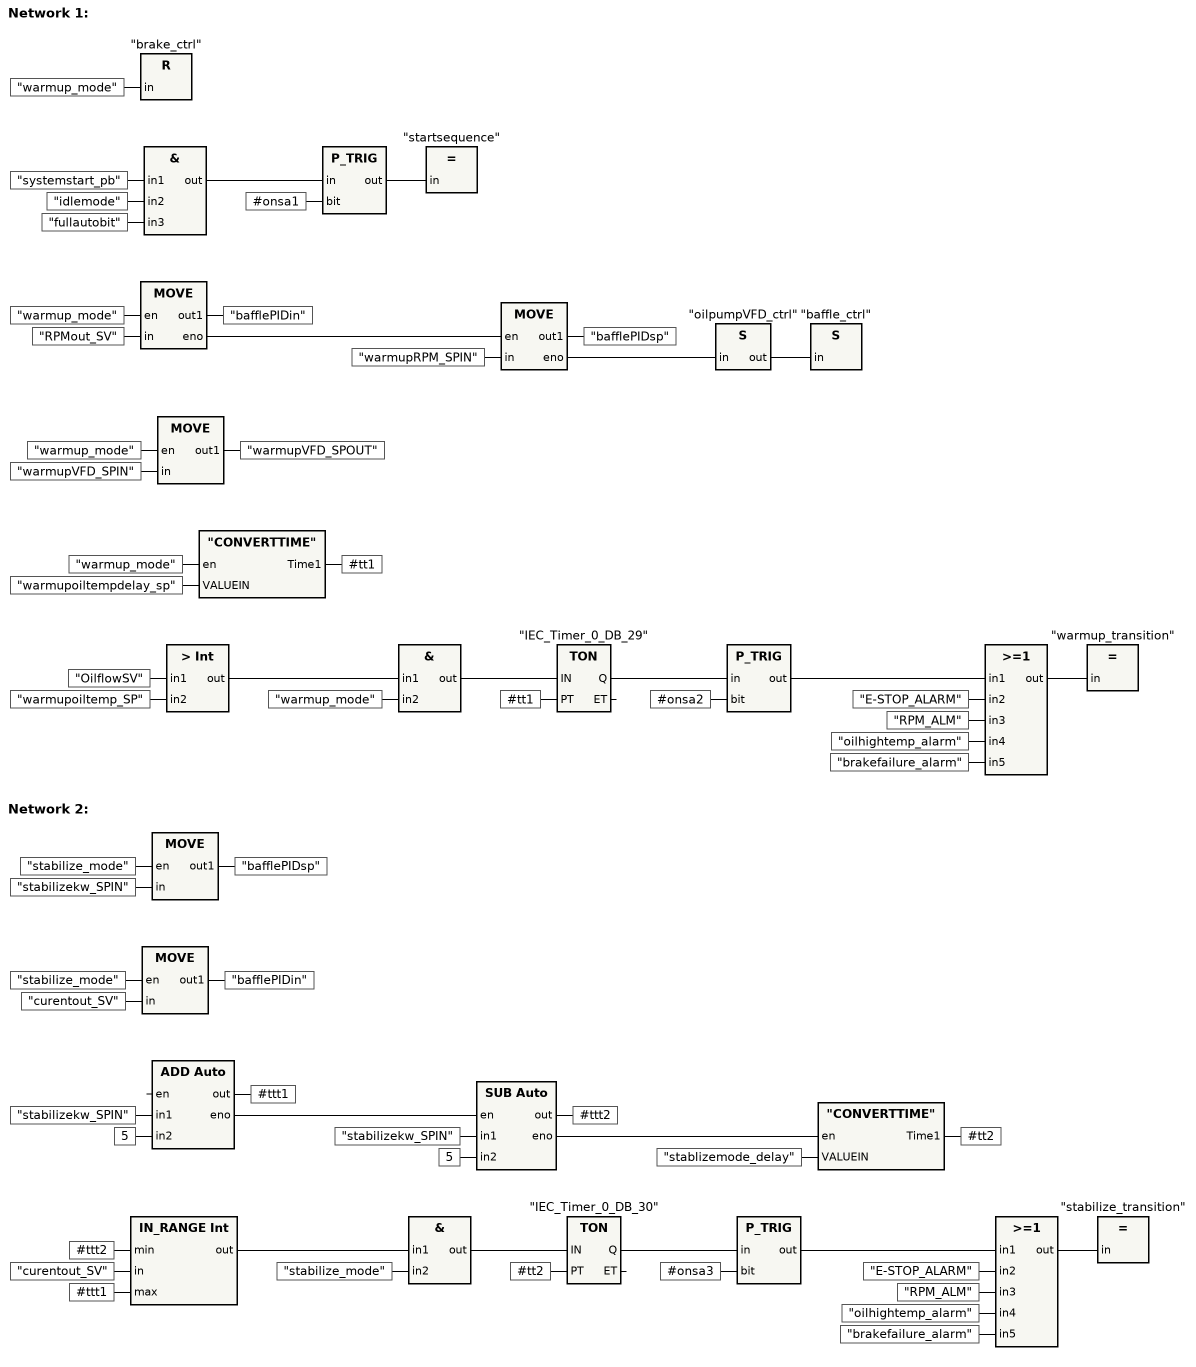
   IF "warmup_mode" THEN "brake_ctrl" := FALSE; END_IF;
   #_w1 := "systemstart_pb" AND "idlemode" AND "fullautobit";
   #_w2 := #_w1 AND NOT #onsa1;   // rising edge
   #onsa1 := #_w1;
   "startsequence" := #_w2;
   IF "warmup_mode" THEN
       "bafflePIDin" := "RPMout_SV";
       "bafflePIDsp" := "warmupRPM_SPIN";
       "oilpumpVFD_ctrl" := TRUE;
       "baffle_ctrl" := TRUE;
       "warmupVFD_SPOUT" := "warmupVFD_SPIN";
       "CONVERTTIME"(VALUEIN := "warmupoiltempdelay_sp", Time1 => #tt1);
   END_IF;
   "IEC_Timer_0_DB_29".TON(IN := ("OilflowSV" > "warmupoiltemp_SP") AND "warmup_mode", PT := #tt1);
   #_w3 := "IEC_Timer_0_DB_29".Q AND NOT #onsa2;   // rising edge
   #onsa2 := "IEC_Timer_0_DB_29".Q;
   "warmup_transition" := #_w3 OR "E-STOP_ALARM" OR "RPM_ALM" OR "oilhightemp_alarm" OR "brakefailure_alarm";
END_REGION

REGION Network 2
   // stability_mode
   IF "stabilize_mode" THEN
       "bafflePIDsp" := "stabilizekw_SPIN";
       "bafflePIDin" := "curentout_SV";
   END_IF;
   #ttt1 := "stabilizekw_SPIN" + 5;
   #ttt2 := "stabilizekw_SPIN" - 5;
   "CONVERTTIME"(VALUEIN := "stablizemode_delay", Time1 => #tt2);
   "IEC_Timer_0_DB_30".TON(IN := (#ttt2 <= "curentout_SV") AND ("curentout_SV" <= #ttt1) AND "stabilize_mode",
                           PT := #tt2);
   #_w1 := "IEC_Timer_0_DB_30".Q AND NOT #onsa3;   // rising edge
   #onsa3 := "IEC_Timer_0_DB_30".Q;
   "stabilize_transition" := #_w1 OR "E-STOP_ALARM" OR "RPM_ALM" OR "oilhightemp_alarm" OR "brakefailure_alarm";
END_REGION

REGION Network 3
   // generation_mode
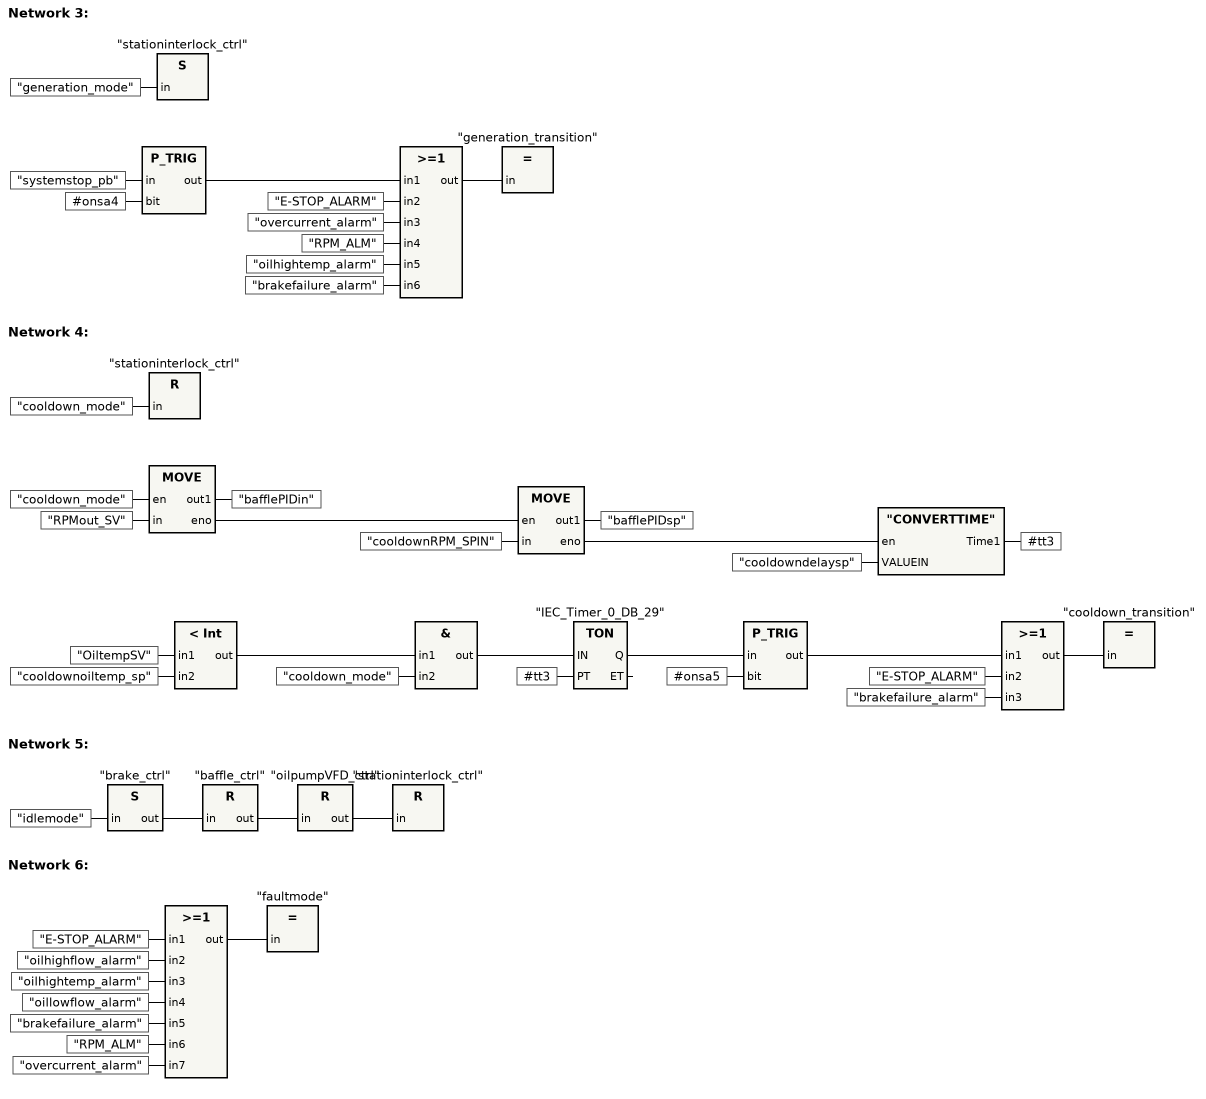
   IF "generation_mode" THEN "stationinterlock_ctrl" := TRUE; END_IF;
   #_w1 := "systemstop_pb" AND NOT #onsa4;   // rising edge
   #onsa4 := "systemstop_pb";
   "generation_transition" := #_w1 OR "E-STOP_ALARM" OR "overcurrent_alarm" OR "RPM_ALM" OR "oilhightemp_alarm" OR "brakefailure_alarm";
END_REGION

REGION Network 4
   // cool_mode
   IF "cooldown_mode" THEN
       "stationinterlock_ctrl" := FALSE;
       "bafflePIDin" := "RPMout_SV";
       "bafflePIDsp" := "cooldownRPM_SPIN";
       "CONVERTTIME"(VALUEIN := "cooldowndelaysp", Time1 => #tt3);
   END_IF;
   "IEC_Timer_0_DB_29".TON(IN := ("OiltempSV" < "cooldownoiltemp_sp") AND "cooldown_mode", PT := #tt3);
   #_w1 := "IEC_Timer_0_DB_29".Q AND NOT #onsa5;   // rising edge
   #onsa5 := "IEC_Timer_0_DB_29".Q;
   "cooldown_transition" := #_w1 OR "E-STOP_ALARM" OR "brakefailure_alarm";
END_REGION

REGION Network 5
   // idlemode
   IF "idlemode" THEN
       "brake_ctrl" := TRUE;
       "baffle_ctrl" := FALSE;
       "oilpumpVFD_ctrl" := FALSE;
       "stationinterlock_ctrl" := FALSE;
   END_IF;
END_REGION

REGION Network 6
   // faultmode
   "faultmode" := "E-STOP_ALARM" OR "oilhighflow_alarm" OR "oilhightemp_alarm" OR "oillowflow_alarm" OR "brakefailure_alarm" OR "RPM_ALM" OR "overcurrent_alarm";
END_REGION
END_FUNCTION_BLOCK

FUNCTION_BLOCK "MODES_SCL"   // FB16, SCL
{ S7_Optimized_Access := 'TRUE' }
VERSION : 0.1
   VAR
      warmuptransitiontrigger : Bool;
      trigger2 : Bool;
      trigger3 : Bool;
   END_VAR
   VAR_TEMP
      tt1 : Time;
      t11 : Time;
      tv1 : Int;
      tv2 : Int;
      tt2 : Time;
      t111 : Time;
      tt3 : Time;
      ttt1 : Time;
   END_VAR
BEGIN
   //ESTOP ALRM
   IF "E-STOP_ALARM" OR "brakefailure_alarm" THEN
       "warmup_transition" := 1;
       "stabilize_transition" := 1;
       "generation_transition" := 1;
       "cooldown_transition" := 1;
   ELSE
       "warmup_transition" := 0;
       "stabilize_transition" := 0;
       "generation_transition" := 0;
       "cooldown_transition" := 0;

       //warmup mode
       IF "systemstart_pb" AND "idlemode" AND "fullautobit" THEN
           "startsequence" := 1;
       ELSE
           "startsequence" := 0;
       END_IF;

       IF "warmup_mode" THEN
           "bafflePIDin" := "RPMout_SV";
           "bafflePIDsp" := "warmupRPM_SPIN";
           "baffle_ctrl" := 1;
           "oilpumpVFD_ctrl" := 1;
           "brake_ctrl" := 0;
           "warmupVFD_SPOUT" := "warmupVFD_SPIN";


           IF "OiltempSV" > "warmupoiltemp_SP" THEN
               "CONVERTTIME"(VALUEIN := "warmupoiltempdelay_sp",
                             Time1 => #tt1);
               "IEC_Timer_0_DB_31".TON(IN := TRUE,
                                       PT := #tt1,
                                       Q => #warmuptransitiontrigger,
                                       ET => #t11);
           ELSE
               RESET_TIMER("IEC_Timer_0_DB_31");
           END_IF;
           IF #warmuptransitiontrigger AND NOT "warmup_transition" THEN
               RESET_TIMER("IEC_Timer_0_DB_31");

               "warmup_transition" := 1;
           END_IF;
       ELSE
           "warmup_transition" := 0;
       END_IF;
       IF "RPM_ALM" OR "oilhightemp_alarm" THEN
           "warmup_transition" := 1;
       END_IF;
       //stabilize_mod
       IF "stabilize_mode" THEN
           "bafflePIDin" := "curentout_SV";
           "bafflePIDsp" := "stabilizekw_SPIN";
           #tv1 := "stabilizekw_SPIN" - 5;
           #tv2 := "stabilizekw_SPIN" + 5;
           IF "curentout_SV" < #tv2 AND "curentout_SV" > #tv1 THEN
               "CONVERTTIME"(VALUEIN := "stablizemode_delay",
                             Time1 => #tt2);
               "IEC_Timer_0_DB_32".TON(IN := TRUE,
                                       PT := #tt2,
                                       Q => #trigger2,
                                       ET => #t111);
           END_IF;
           IF #trigger2 AND NOT "stabilize_transition" THEN
               RESET_TIMER("IEC_Timer_0_DB_32");

               "stabilize_transition" := 1;
           END_IF;
       ELSE
           "stabilize_transition" := 0;
       END_IF;
       IF "RPM_ALM" OR "oilhightemp_alarm" THEN
           "stabilize_transition" := 1;
       END_IF;

       //generation_mode
       IF "generation_mode" THEN
           "stationinterlock_ctrl" := 1;


           IF "systemstop_pb" AND NOT "generation_transition" THEN
               "generation_transition" := 1;
           END_IF;
       ELSE
           "generation_transition" := 0;
       END_IF;

       IF "overcurrent_alarm" OR "RPM_ALM" OR "oilhightemp_alarm" THEN
           "generation_transition" := 1;
       END_IF;

       //coolmode
       IF "cooldown_mode" THEN
           "stationinterlock_ctrl" := 0;
           "bafflePIDin" := "RPMout_SV";
           "bafflePIDsp" := "cooldownRPM_SPIN";

           IF "OiltempSV" < "cooldownoiltemp_sp" THEN
               "CONVERTTIME"(VALUEIN := "cooldowndelaysp",
                             Time1 => #tt3);
               "IEC_Timer_0_DB_33".TON(IN := TRUE,
                                       PT := #tt3,
                                       Q => #trigger3,
                                       ET => #ttt1);

           END_IF;
           IF #trigger3 AND NOT "idlemode_transition" THEN
               RESET_TIMER("IEC_Timer_0_DB_33");

               "cooldown_transition" := 1;
           END_IF;
       ELSE
           "cooldown_transition" := 0;
       END_IF;

       //idlemode
       IF "idlemode" THEN
           "brake_ctrl" := 1;
           "baffle_ctrl" := 0;
           "oilpumpVFD_ctrl" := 0;

       END_IF;

       //faultmode

       IF "E-STOP_ALARM" OR "oilhighflow_alarm" OR "oillowflow_alarm" OR "oilhightemp_alarm" OR "brakefailure_alarm" OR "overcurrent_alarm" OR "RPM_ALM" THEN
           "faultmode" := 1;
       ELSE
           "faultmode" := 0;
       END_IF;


   END_IF;
   //idlemode
   IF "idlemode" THEN
       "brake_ctrl" := 1;
       "baffle_ctrl" := 0;
       "oilpumpVFD_ctrl" := 0;
       "stationinterlock_ctrl" := 0;

   END_IF;
END_FUNCTION_BLOCK

FUNCTION_BLOCK "MODES_STL"   // FB17, STL
{ S7_Optimized_Access := 'TRUE' }
VERSION : 0.1
   VAR
      trigger1 : Bool;
      ONSA1 : Bool;
      OS2 : Bool;
      ONS : Bool;
   END_VAR
   VAR_TEMP
      tv1 : Time;
      t1v1 : Time;
      ttv1 : Int;
      ttv2 : Int;
      tttv2 : Int;
      tb1 : Bool;
      tv2 : Time;
      trigger2 : Bool;
      tt2 : Time;
      onsa2 : Bool;
      tv3 : Time;
      trigger3 : Bool;
      ttt4 : Time;
   END_VAR
BEGIN

REGION Network 1
   //ESTOP HANDLING
         A     "E-STOP_ALARM";
         O     "brakefailure_alarm";
         JC    ESTOPTRANSITION;
         JU    resettransition;


   ESTOPTRANSITION:SET;
         S     "warmup_transition";
         S     "stabilize_transition";
         S     "generation_transition";
         S     "cooldown_transition";
         JU    JUMPTOMODE;

   resettransition:CLR;
         NOT;
         R     "warmup_transition";
         R     "stabilize_transition";
         R     "generation_transition";
         R     "cooldown_transition";
         R     "startsequence";

   JUMPTOMODE:A     "warmup_mode";
         JC    startwarmupmode;
         CLR;
         A     "stabilize_mode";
         JC    stabilizemode;
         CLR;
         A     "generation_mode";
         JC    generationmode;
         CLR;
         A     "cooldown_mode";
         JC    cooldownmode;
         CLR;
         A     "idlemode";
         JC    idlemode;
         JU    faultmode;


   // WARMMODE



   startwarmupmode:R     "brake_ctrl";
         L     "warmupRPM_SPIN";
         T     "bafflePIDsp";
         L     "RPMout_SV";
         T     "bafflePIDin";


         SET;
         S     "oilpumpVFD_ctrl";
         S     "baffle_ctrl";
         L     "warmupVFD_SPIN";
         L     "warmupVFD_SPOUT";

         L     "OiltempSV";
         L     "warmupoiltemp_SP";
         >I;
         JC    warmuptime;
         CALL  RESET_TIMER
         ( "TIMER" := "IEC_Timer_0_DB_34"
         );

         JU    stabilizemode;

   warmuptime:CALL  "CONVERTTIME"
         ( VALUEIN := "warmupoiltempdelay_sp",
           Time1   := #tv1
         );
         CALL  TON, "IEC_Timer_0_DB_34"
         ( IN := true,
           PT := #tv1,
           Q  := #trigger1,
           ET := #t1v1
         );

         A     #trigger1;

         JC    warmtimer;
         CLR;
         A     "RPM_ALM";
         O     "oilhighflow_alarm";
         JC    warmtimer;

         JU    stabilizemode;
   warmtimer:S     "warmup_transition";
         CALL  RESET_TIMER
         ( "TIMER" := "IEC_Timer_0_DB_34"
         );
         JU    stabilizemode;

   // STABILIZE MODE
   stabilizemode:SET;
         NOT;
         R     "warmup_transition";

         L     "curentout_SV";
         T     "bafflePIDin";
         L     "stabilizekw_SPIN";
         T     "bafflePIDsp";
         L     "stabilizekw_SPIN";
         L     5;
         +I;
         T     #ttv1;
         L     "stabilizekw_SPIN";
         L     5;
         -I;
         T     #ttv2;
         L     "curentout_SV";
         L     #ttv1;
         <I;
         S     #tb1;
         L     "curentout_SV";
         L     #ttv2;
         >I;
         A     #tb1;
         JC    stabilizetime;
         CALL  RESET_TIMER
         ( "TIMER" := "IEC_Timer_0_DB_35"
         );
         JU    generationmode;
   stabilizetime:CALL  "CONVERTTIME"
         ( VALUEIN := "stablizemode_delay",
           Time1   := #tv2
         );

         CALL  TON, "IEC_Timer_0_DB_35"
         ( IN := true,
           PT := #tv2,
           Q  := #trigger2,
           ET := #tt2
         );

         A     #trigger2;

         JC    resetstabilizetimer;
         CLR;
         A     "RPM_ALM";
         O     "oilhighflow_alarm";
         JC    resetstabilizetimer;

         JU    generationmode;
   resetstabilizetimer:S     "stabilize_transition";
         CALL  RESET_TIMER
         ( "TIMER" := "IEC_Timer_0_DB_35"
         );
         JU    generationmode;

   //generationmode
   generationmode:SET;
         NOT;
         R     "stabilize_transition";
         SET;
         S     "stationinterlock_ctrl";

         A     "systemstop_pb";
         JC    generationexit;
         CLR;
         A     "overcurrent_alarm";
         JC    generationexit;
         CLR;
         A     "RPM_ALM";
         O     "oilhighflow_alarm";
         JC    generationexit;
         CLR;

         JU    cooldownmode;

   generationexit:S     "generation_transition";
         JU    cooldownmode;

   //cooldownmode
   cooldownmode:SET;
         NOT;
         R     "generation_transition";
         R     "stationinterlock_ctrl";
         L     "RPMout_SV";
         T     "bafflePIDin";
         L     "cooldownRPM_SPIN";
         T     "bafflePIDsp";
         L     "OiltempSV";
         L     "cooldownoiltemp_sp";
         <I;
         JC    cooldowntimer;

         CALL  RESET_TIMER
         ( "TIMER" := "IEC_Timer_0_DB_36"
         );
         JU    idlemode;
   cooldowntimer:CALL  "CONVERTTIME"
         ( VALUEIN := "cooldowndelaysp",
           Time1   := #tv3
         );
         CALL  TON, "IEC_Timer_0_DB_36"
         ( IN := true,
           PT := #tv3,
           Q  := #trigger3,
           ET := #ttt4
         );
         A     #trigger3;

         JC    resetcooltimer;
         JU    idlemode;
   resetcooltimer:S     "cooldown_transition";
         CALL  RESET_TIMER
         ( "TIMER" := "IEC_Timer_0_DB_36"
         );
         JU    idlemode;

   //idlemode
   idlemode:SET;
         NOT;
         R     "cooldown_transition";
         R     "baffle_ctrl";
         R     "oilpumpVFD_ctrl";
         R     "stationinterlock_ctrl";
         S     "brake_ctrl";
         CLR;
         A     "systemstart_pb";
         A     "idlemode";
         A     "fullautobit";
         FP    #ONS;
         S     "startsequence";

         JU    faultmode;

   //FAULTMODE
   faultmode:A     "E-STOP_ALARM";
         O     "oilhighflow_alarm";
         O     "oillowflow_alarm";
         O     "oilhightemp_alarm";
         O     "brakefailure_alarm";
         O     "overcurrent_alarm";
         O     "RPM_ALM";
         S     "faultmode";
END_REGION
END_FUNCTION_BLOCK

